LIN {X 0,Y 312.174,Z 269.379,A -85,B 0,C 180,E1 -15950.08,E2 -15950.08} C_VEL
LIN {X 0,Y 314.223,Z 258.273,A -85,B 0,C 180,E1 -15951.484,E2 -15951.484} C_VEL
LIN {X 0,Y 316.003,Z 247.419,A -85,B 0,C 180,E1 -15952.56,E2 -15952.56} C_VEL
LIN {X 0,Y 317.612,Z 235.462,A -85,B 0,C 180,E1 -15953.472,E2 -15953.472} C_VEL
LIN {X 0,Y 318.995,Z 222.423,A -85,B 0,C 180,E1 -15954.183,E2 -15954.183} C_VEL
LIN {X 0,Y 319.798,Z 209.498,A -85,B 0,C 180,E1 -15954.637,E2 -15954.637} C_VEL
LIN {X 0,Y 321.419,Z 151.601,A -85,B 0,C 180,E1 -15955.948,E2 -15955.948} C_VEL
LIN {X 0,Y 317.976,Z 130.29,A -85,B 0,C 180,E1 -15956.843,E2 -15956.843} C_VEL
LIN {X 0,Y 313.089,Z 106.225,A -85,B 0,C 180,E1 -15957.999,E2 -15957.999} C_VEL
LIN {X 0,Y 312.175,Z 103.135,A -85,B 0,C 180,E1 -15958.215,E2 -15958.215} C_VEL
LIN {X 0,Y 309.987,Z 92.53,A -85,B 0,C 180,E1 -15961.43,E2 -15961.43} C_VEL
LIN {X 0,Y 307.446,Z 81.962,A -85,B 0,C 180,E1 -15964.854,E2 -15964.854} C_VEL
LIN {X 0,Y 305.474,Z 74.435,A -85,B 0,C 180,E1 -15967.463,E2 -15967.463} C_VEL
LIN {X 0,Y 305.457,Z 74.429,A -85,B 0,C 180,E1 -15970.6,E2 -15970.6} C_VEL
LIN {X 0,Y 305.428,Z 74.438,A -85,B 0,C 180,E1 -15973.655,E2 -15973.655} C_VEL
LIN {X 0,Y 305.457,Z 74.427,A -85,B 0,C 180,E1 -15977.414,E2 -15977.414} C_VEL
LIN {X 0,Y 305.478,Z 74.431,A -85,B 0,C 180,E1 -15981.598,E2 -15981.598} C_VEL
LIN {X 0,Y 305.465,Z 74.433,A -85,B 0,C 180,E1 -15984.887,E2 -15984.887} C_VEL
LIN {X 0,Y 305.455,Z 74.435,A -85,B 0,C 180,E1 -15988.355,E2 -15988.355} C_VEL
LIN {X 0,Y 305.523,Z 74.424,A -85,B 0,C 180,E1 -15991.114,E2 -15991.114} C_VEL
LIN {X 0,Y 305.574,Z 74.412,A -85,B 0,C 180,E1 -15994.088,E2 -15994.088} C_VEL
LIN {X 0,Y 305.503,Z 74.421,A -85,B 0,C 180,E1 -15998.403,E2 -15998.403} C_VEL
LIN {X 0,Y 305.593,Z 74.417,A -85,B 0,C 180,E1 -16001.218,E2 -16001.218} C_VEL
LIN {X 0,Y 305.652,Z 74.41,A -85,B 0,C 180,E1 -16005.349,E2 -16005.349} C_VEL
LIN {X 0,Y 305.639,Z 74.409,A -85,B 0,C 180,E1 -16009.4,E2 -16009.4} C_VEL
LIN {X 0,Y 305.8,Z 74.385,A -85,B 0,C 180,E1 -16012.074,E2 -16012.074} C_VEL
LIN {X 0,Y 305.687,Z 74.406,A -85,B 0,C 180,E1 -16014.723,E2 -16014.723} C_VEL
LIN {X 0,Y 305.958,Z 74.362,A -85,B 0,C 180,E1 -16018.684,E2 -16018.684} C_VEL
LIN {X 0,Y 305.959,Z 74.374,A -85,B 0,C 180,E1 -16021.316,E2 -16021.316} C_VEL
LIN {X 0,Y 305.684,Z 74.403,A -85,B 0,C 180,E1 -16025.276,E2 -16025.276} C_VEL
LIN {X 0,Y 305.774,Z 74.388,A -85,B 0,C 180,E1 -16027.927,E2 -16027.927} C_VEL
LIN {X 0,Y 305.602,Z 74.416,A -85,B 0,C 180,E1 -16031.945,E2 -16031.945} C_VEL
LIN {X 0,Y 305.611,Z 74.41,A -85,B 0,C 180,E1 -16035.014,E2 -16035.014} C_VEL
LIN {X 0,Y 305.563,Z 74.417,A -85,B 0,C 180,E1 -16039.437,E2 -16039.437} C_VEL
LIN {X 0,Y 305.49,Z 74.424,A -85,B 0,C 180,E1 -16043.04,E2 -16043.04} C_VEL
LIN {X 0,Y 305.48,Z 74.431,A -85,B 0,C 180,E1 -16046.2,E2 -16046.2} C_VEL
LIN {X 0,Y 305.465,Z 74.436,A -85,B 0,C 180,E1 -16049.039,E2 -16049.039} C_VEL
LIN {X 0,Y 305.438,Z 74.437,A -85,B 0,C 180,E1 -16051.953,E2 -16051.953} C_VEL
LIN {X 0,Y 305.463,Z 74.436,A -85,B 0,C 180,E1 -16055.113,E2 -16055.113} C_VEL
LIN {X 0,Y 305.436,Z 74.44,A -85,B 0,C 180,E1 -16058.525,E2 -16058.525} C_VEL
LIN {X 0,Y 305.44,Z 74.426,A -85,B 0,C 180,E1 -16061.857,E2 -16061.857} C_VEL
LIN {X 0,Y 305.401,Z 74.447,A -85,B 0,C 180,E1 -16065.511,E2 -16065.511} C_VEL
LIN {X 0,Y 305.44,Z 74.438,A -85,B 0,C 180,E1 -16068.143,E2 -16068.143} C_VEL
LIN {X 0,Y 305.469,Z 74.592,A -85,B 0,C 180,E1 -16070.734,E2 -16070.734} C_VEL
LIN {X 0,Y 305.694,Z 75.552,A -85,B 0,C 180,E1 -16071.094,E2 -16071.094} C_VEL
LIN {X 0,Y 315.489,Z 94.618,A -85,B 0,C 180,E1 -16072.75,E2 -16072.75} C_VEL
LIN {X 0,Y 322.655,Z 110.769,A -85,B 0,C 180,E1 -16073.933,E2 -16073.933} C_VEL
LIN {X 0,Y 320.349,Z 182.482,A -85,B 0,C 180,E1 -16075.556,E2 -16075.556} C_VEL
LIN {X 0,Y 319.573,Z 195.788,A -85,B 0,C 180,E1 -16076.127,E2 -16076.127} C_VEL
LIN {X 0,Y 318.63,Z 208.433,A -85,B 0,C 180,E1 -16076.947,E2 -16076.947} C_VEL
LIN {X 0,Y 317.275,Z 219.431,A -85,B 0,C 180,E1 -16077.884,E2 -16077.884} C_VEL
LIN {X 0,Y 315.483,Z 231.187,A -85,B 0,C 180,E1 -16079.178,E2 -16079.178} C_VEL
LIN {X 0,Y 313.661,Z 241.965,A -85,B 0,C 180,E1 -16080.695,E2 -16080.695} C_VEL
LIN {X 0,Y 311.646,Z 251.896,A -85,B 0,C 180,E1 -16082.464,E2 -16082.464} C_VEL
LIN {X 0,Y 309.803,Z 260.794,A -85,B 0,C 180,E1 -16084.467,E2 -16084.467} C_VEL
LIN {X 0,Y 308.194,Z 267.818,A -85,B 0,C 180,E1 -16086.48,E2 -16086.48} C_VEL
LIN {X 0,Y 306.828,Z 273.393,A -85,B 0,C 180,E1 -16088.501,E2 -16088.501} C_VEL
LIN {X 0,Y 305.902,Z 277.442,A -85,B 0,C 180,E1 -16090.384,E2 -16090.384} C_VEL
LIN {X 0,Y 304.998,Z 280.942,A -85,B 0,C 180,E1 -16092.569,E2 -16092.569} C_VEL
LIN {X 0,Y 304.582,Z 282.525,A -85,B 0,C 180,E1 -16093.925,E2 -16093.925} C_VEL
LIN {X 0,Y 304.153,Z 284.125,A -85,B 0,C 180,E1 -16096.044,E2 -16096.044} C_VEL
LIN {X 0,Y 303.866,Z 284.702,A -85,B 0,C 180,E1 -16097.986,E2 -16097.986} C_VEL
LIN {X 0,Y 303.732,Z 284.63,A -85,B 0,C 180,E1 -16099.332,E2 -16099.332} C_VEL
LIN {X 0,Y 303.757,Z 284.146,A -85,B 0,C 180,E1 -16100.679,E2 -16100.679} C_VEL
LIN {X 0,Y 303.995,Z 281.922,A -85,B 0,C 180,E1 -16103.362,E2 -16103.362} C_VEL
LIN {X 0,Y 304.17,Z 279.182,A -85,B 0,C 180,E1 -16105.362,E2 -16105.362} C_VEL
LIN {X 0,Y 304.546,Z 275.426,A -85,B 0,C 180,E1 -16107.355,E2 -16107.355} C_VEL
LIN {X 0,Y 304.948,Z 270.574,A -85,B 0,C 180,E1 -16109.34,E2 -16109.34} C_VEL
LIN {X 0,Y 305.686,Z 264.452,A -85,B 0,C 180,E1 -16111.318,E2 -16111.318} C_VEL
LIN {X 0,Y 306.662,Z 256.84,A -85,B 0,C 180,E1 -16113.285,E2 -16113.285} C_VEL
LIN {X 0,Y 307.747,Z 247.299,A -85,B 0,C 180,E1 -16115.241,E2 -16115.241} C_VEL
LIN {X 0,Y 308.92,Z 238.487,A -85,B 0,C 180,E1 -16116.696,E2 -16116.696} C_VEL
LIN {X 0,Y 310.231,Z 227.693,A -85,B 0,C 180,E1 -16118.14,E2 -16118.14} C_VEL
LIN {X 0,Y 311.278,Z 217.16,A -85,B 0,C 180,E1 -16119.257,E2 -16119.257} C_VEL
LIN {X 0,Y 312.202,Z 204.544,A -85,B 0,C 180,E1 -16120.293,E2 -16120.293} C_VEL
LIN {X 0,Y 312.857,Z 191.92,A -85,B 0,C 180,E1 -16121.049,E2 -16121.049} C_VEL
LIN {X 0,Y 313.315,Z 179.752,A -85,B 0,C 180,E1 -16121.524,E2 -16121.524} C_VEL
LIN {X 0,Y 314.897,Z 100.853,A -85,B 0,C 180,E1 -16123.325,E2 -16123.325} C_VEL
LIN {X 0,Y 307.555,Z 79.529,A -85,B 0,C 180,E1 -16124.348,E2 -16124.348} C_VEL
LIN {X 0,Y 305.659,Z 74.413,A -85,B 0,C 180,E1 -16124.624,E2 -16124.624} C_VEL
LIN {X 0,Y 305.591,Z 74.419,A -85,B 0,C 180,E1 -16128.783,E2 -16128.783} C_VEL
LIN {X 0,Y 305.487,Z 74.43,A -85,B 0,C 180,E1 -16133.04,E2 -16133.04} C_VEL
LIN {X 0,Y 305.548,Z 74.427,A -85,B 0,C 180,E1 -16136.227,E2 -16136.227} C_VEL
LIN {X 0,Y 305.489,Z 74.43,A -85,B 0,C 180,E1 -16139.048,E2 -16139.048} C_VEL
LIN {X 0,Y 305.445,Z 74.44,A -85,B 0,C 180,E1 -16141.952,E2 -16141.952} C_VEL
LIN {X 0,Y 305.465,Z 74.433,A -85,B 0,C 180,E1 -16145.113,E2 -16145.113} C_VEL
LIN {X 0,Y 305.469,Z 74.432,A -85,B 0,C 180,E1 -16148.533,E2 -16148.533} C_VEL
LIN {X 0,Y 305.475,Z 74.431,A -85,B 0,C 180,E1 -16152.59,E2 -16152.59} C_VEL
LIN {X 0,Y 305.457,Z 74.438,A -85,B 0,C 180,E1 -16157.415,E2 -16157.415} C_VEL
LIN {X 0,Y 305.442,Z 74.436,A -85,B 0,C 180,E1 -16159.149,E2 -16159.149} C_VEL
LIN {X 0,Y 304.808,Z 74.519,A -85,B 0,C 180,E1 -16160.25,E2 -16160.25} C_VEL
LIN {X 0,Y 301.942,Z 74.872,A -85,B 0,C 180,E1 -16162.043,E2 -16162.043} C_VEL
LIN {X 0,Y 299.502,Z 75.176,A -85,B 0,C 180,E1 -16163.497,E2 -16163.497} C_VEL
LIN {X 0,Y 298.474,Z 75.302,A -85,B 0,C 180,E1 -16164.624,E2 -16164.624} C_VEL
LIN {X 0,Y 298.402,Z 75.309,A -85,B 0,C 180,E1 -16165.006,E2 -16165.006} C_VEL
LIN {X 0,Y 298.395,Z 75.316,A -85,B 0,C 180,E1 -16168.791,E2 -16168.791} C_VEL
LIN {X 0,Y 298.462,Z 75.305,A -85,B 0,C 180,E1 -16171.904,E2 -16171.904} C_VEL
LIN {X 0,Y 298.489,Z 75.304,A -85,B 0,C 180,E1 -16174.924,E2 -16174.924} C_VEL
LIN {X 0,Y 298.454,Z 75.305,A -85,B 0,C 180,E1 -16179.316,E2 -16179.316} C_VEL
LIN {X 0,Y 298.541,Z 75.293,A -85,B 0,C 180,E1 -16182.18,E2 -16182.18} C_VEL
LIN {X 0,Y 298.597,Z 75.284,A -85,B 0,C 180,E1 -16184.995,E2 -16184.995} C_VEL
LIN {X 0,Y 298.587,Z 75.289,A -85,B 0,C 180,E1 -16189.147,E2 -16189.147} C_VEL
LIN {X 0,Y 298.736,Z 75.273,A -85,B 0,C 180,E1 -16191.885,E2 -16191.885} C_VEL
LIN {X 0,Y 298.657,Z 75.273,A -85,B 0,C 180,E1 -16194.599,E2 -16194.599} C_VEL
LIN {X 0,Y 298.926,Z 75.245,A -85,B 0,C 180,E1 -16198.653,E2 -16198.653} C_VEL
LIN {X 0,Y 298.926,Z 75.248,A -85,B 0,C 180,E1 -16201.347,E2 -16201.347} C_VEL
LIN {X 0,Y 298.643,Z 75.283,A -85,B 0,C 180,E1 -16205.402,E2 -16205.402} C_VEL
LIN {X 0,Y 298.712,Z 75.274,A -85,B 0,C 180,E1 -16208.116,E2 -16208.116} C_VEL
LIN {X 0,Y 298.554,Z 75.293,A -85,B 0,C 180,E1 -16212.232,E2 -16212.232} C_VEL
LIN {X 0,Y 298.553,Z 75.297,A -85,B 0,C 180,E1 -16215.169,E2 -16215.169} C_VEL
LIN {X 0,Y 298.524,Z 75.3,A -85,B 0,C 180,E1 -16219.244,E2 -16219.244} C_VEL
LIN {X 0,Y 298.429,Z 75.31,A -85,B 0,C 180,E1 -16223.6,E2 -16223.6} C_VEL
LIN {X 0,Y 298.42,Z 75.313,A -85,B 0,C 180,E1 -16226.581,E2 -16226.581} C_VEL
LIN {X 0,Y 298.403,Z 75.313,A -85,B 0,C 180,E1 -16229.643,E2 -16229.643} C_VEL
LIN {X 0,Y 298.396,Z 75.318,A -85,B 0,C 180,E1 -16232.8,E2 -16232.8} C_VEL
LIN {X 0,Y 298.45,Z 75.31,A -85,B 0,C 180,E1 -16236.808,E2 -16236.808} C_VEL
LIN {X 0,Y 298.39,Z 75.315,A -85,B 0,C 180,E1 -16241.088,E2 -16241.088} C_VEL
LIN {X 0,Y 298.401,Z 75.312,A -85,B 0,C 180,E1 -16243.103,E2 -16243.103} C_VEL
LIN {X 0,Y 298.406,Z 75.313,A -85,B 0,C 180,E1 -16246.921,E2 -16246.921} C_VEL
LIN {X 0,Y 298.398,Z 75.314,A -85,B 0,C 180,E1 -16251.008,E2 -16251.008} C_VEL
LIN {X 0,Y 298.419,Z 75.312,A -85,B 0,C 180,E1 -16253.93,E2 -16253.93} C_VEL
LIN {X 0,Y 298.459,Z 75.446,A -85,B 0,C 180,E1 -16257.157,E2 -16257.157} C_VEL
LIN {X 0,Y 301.343,Z 88.771,A -85,B 0,C 180,E1 -16261.057,E2 -16261.057} C_VEL
LIN {X 0,Y 302.506,Z 95.962,A -85,B 0,C 180,E1 -16263.061,E2 -16263.061} C_VEL
LIN {X 0,Y 301.566,Z 103.824,A -85,B 0,C 180,E1 -16265.076,E2 -16265.076} C_VEL
LIN {X 0,Y 306.342,Z 141.137,A -85,B 0,C 180,E1 -16266.335,E2 -16266.335} C_VEL
LIN {X 0,Y 307.368,Z 151.276,A -85,B 0,C 180,E1 -16266.651,E2 -16266.651} C_VEL
LIN {X 0,Y 306.075,Z 212.628,A -85,B 0,C 180,E1 -16268.091,E2 -16268.091} C_VEL
LIN {X 0,Y 305.295,Z 225.998,A -85,B 0,C 180,E1 -16268.653,E2 -16268.653} C_VEL
LIN {X 0,Y 304.267,Z 238.814,A -85,B 0,C 180,E1 -16269.463,E2 -16269.463} C_VEL
LIN {X 0,Y 302.972,Z 250.972,A -85,B 0,C 180,E1 -16270.521,E2 -16270.521} C_VEL
LIN {X 0,Y 301.528,Z 262.552,A -85,B 0,C 180,E1 -16271.835,E2 -16271.835} C_VEL
LIN {X 0,Y 300.343,Z 273.016,A -85,B 0,C 180,E1 -16273.342,E2 -16273.342} C_VEL
LIN {X 0,Y 299.404,Z 281.24,A -85,B 0,C 180,E1 -16274.799,E2 -16274.799} C_VEL
LIN {X 0,Y 298.344,Z 290.113,A -85,B 0,C 180,E1 -16276.722,E2 -16276.722} C_VEL
LIN {X 0,Y 297.419,Z 297.659,A -85,B 0,C 180,E1 -16278.758,E2 -16278.758} C_VEL
LIN {X 0,Y 296.928,Z 304.631,A -85,B 0,C 180,E1 -16281.15,E2 -16281.15} C_VEL
LIN {X 0,Y 296.642,Z 309.207,A -85,B 0,C 180,E1 -16283.197,E2 -16283.197} C_VEL
LIN {X 0,Y 296.641,Z 311.618,A -85,B 0,C 180,E1 -16284.562,E2 -16284.562} C_VEL
LIN {X 0,Y 296.692,Z 313.588,A -85,B 0,C 180,E1 -16285.925,E2 -16285.925} C_VEL
LIN {X 0,Y 296.691,Z 315.127,A -85,B 0,C 180,E1 -16287.284,E2 -16287.284} C_VEL
LIN {X 0,Y 296.759,Z 316.208,A -85,B 0,C 180,E1 -16288.643,E2 -16288.643} C_VEL
LIN {X 0,Y 296.843,Z 316.882,A -85,B 0,C 180,E1 -16290,E2 -16290} C_VEL
LIN {X 0,Y 296.624,Z 317.031,A -85,B 0,C 180,E1 -16292.716,E2 -16292.716} C_VEL
LIN {X 0,Y 296.597,Z 316.486,A -85,B 0,C 180,E1 -16294.076,E2 -16294.076} C_VEL
LIN {X 0,Y 296.646,Z 314.191,A -85,B 0,C 180,E1 -16296.803,E2 -16296.803} C_VEL
LIN {X 0,Y 296.972,Z 311.382,A -85,B 0,C 180,E1 -16298.849,E2 -16298.849} C_VEL
LIN {X 0,Y 297.529,Z 307.567,A -85,B 0,C 180,E1 -16300.893,E2 -16300.893} C_VEL
LIN {X 0,Y 298.461,Z 302.656,A -85,B 0,C 180,E1 -16302.926,E2 -16302.926} C_VEL
LIN {X 0,Y 299.869,Z 296.503,A -85,B 0,C 180,E1 -16304.94,E2 -16304.94} C_VEL
LIN {X 0,Y 301.468,Z 289.016,A -85,B 0,C 180,E1 -16306.909,E2 -16306.909} C_VEL
LIN {X 0,Y 303.08,Z 281.127,A -85,B 0,C 180,E1 -16308.593,E2 -16308.593} C_VEL
LIN {X 0,Y 305.307,Z 270.619,A -85,B 0,C 180,E1 -16310.375,E2 -16310.375} C_VEL
LIN {X 0,Y 307.451,Z 259.953,A -85,B 0,C 180,E1 -16311.806,E2 -16311.806} C_VEL
LIN {X 0,Y 309.207,Z 249.659,A -85,B 0,C 180,E1 -16312.907,E2 -16312.907} C_VEL
LIN {X 0,Y 311.029,Z 237.375,A -85,B 0,C 180,E1 -16313.911,E2 -16313.911} C_VEL
LIN {X 0,Y 312.502,Z 224.487,A -85,B 0,C 180,E1 -16314.674,E2 -16314.674} C_VEL
LIN {X 0,Y 313.425,Z 212.064,A -85,B 0,C 180,E1 -16315.172,E2 -16315.172} C_VEL
LIN {X 0,Y 315.209,Z 152.445,A -85,B 0,C 180,E1 -16316.561,E2 -16316.561} C_VEL
LIN {X 0,Y 311.622,Z 130.195,A -85,B 0,C 180,E1 -16317.528,E2 -16317.528} C_VEL
LIN {X 0,Y 307.049,Z 108.021,A -85,B 0,C 180,E1 -16318.641,E2 -16318.641} C_VEL
LIN {X 0,Y 304.973,Z 102.645,A -85,B 0,C 180,E1 -16319.07,E2 -16319.07} C_VEL
LIN {X 0,Y 302.402,Z 90.76,A -85,B 0,C 180,E1 -16322.837,E2 -16322.837} C_VEL
LIN {X 0,Y 299.638,Z 79.777,A -85,B 0,C 180,E1 -16326.594,E2 -16326.594} C_VEL
LIN {X 0,Y 298.449,Z 75.301,A -85,B 0,C 180,E1 -16328.288,E2 -16328.288} C_VEL
LIN {X 0,Y 298.387,Z 75.316,A -85,B 0,C 180,E1 -16331.261,E2 -16331.261} C_VEL
LIN {X 0,Y 298.356,Z 75.312,A -85,B 0,C 180,E1 -16335.035,E2 -16335.035} C_VEL
LIN {X 0,Y 298.387,Z 75.312,A -85,B 0,C 180,E1 -16338.738,E2 -16338.738} C_VEL
LIN {X 0,Y 298.416,Z 75.307,A -85,B 0,C 180,E1 -16342.242,E2 -16342.242} C_VEL
LIN {X 0,Y 298.411,Z 75.308,A -85,B 0,C 180,E1 -16345.581,E2 -16345.581} C_VEL
LIN {X 0,Y 298.398,Z 75.316,A -85,B 0,C 180,E1 -16348.791,E2 -16348.791} C_VEL
LIN {X 0,Y 298.466,Z 75.306,A -85,B 0,C 180,E1 -16351.904,E2 -16351.904} C_VEL
LIN {X 0,Y 298.489,Z 75.298,A -85,B 0,C 180,E1 -16354.924,E2 -16354.924} C_VEL
LIN {X 0,Y 298.453,Z 75.304,A -85,B 0,C 180,E1 -16359.315,E2 -16359.315} C_VEL
LIN {X 0,Y 298.541,Z 75.29,A -85,B 0,C 180,E1 -16362.179,E2 -16362.179} C_VEL
LIN {X 0,Y 298.597,Z 75.29,A -85,B 0,C 180,E1 -16364.995,E2 -16364.995} C_VEL
LIN {X 0,Y 298.595,Z 75.287,A -85,B 0,C 180,E1 -16369.147,E2 -16369.147} C_VEL
LIN {X 0,Y 298.744,Z 75.266,A -85,B 0,C 180,E1 -16371.885,E2 -16371.885} C_VEL
LIN {X 0,Y 298.658,Z 75.28,A -85,B 0,C 180,E1 -16374.599,E2 -16374.599} C_VEL
LIN {X 0,Y 298.925,Z 75.237,A -85,B 0,C 180,E1 -16378.653,E2 -16378.653} C_VEL
LIN {X 0,Y 298.925,Z 75.25,A -85,B 0,C 180,E1 -16381.347,E2 -16381.347} C_VEL
LIN {X 0,Y 298.778,Z 75.267,A -85,B 0,C 180,E1 -16386.754,E2 -16386.754} C_VEL
LIN {X 0,Y 298.628,Z 75.276,A -85,B 0,C 180,E1 -16389.482,E2 -16389.482} C_VEL
LIN {X 0,Y 298.548,Z 75.285,A -85,B 0,C 180,E1 -16393.615,E2 -16393.615} C_VEL
LIN {X 0,Y 298.49,Z 75.303,A -85,B 0,C 180,E1 -16396.412,E2 -16396.412} C_VEL
LIN {X 0,Y 298.501,Z 75.298,A -85,B 0,C 180,E1 -16399.648,E2 -16399.648} C_VEL
LIN {X 0,Y 298.428,Z 75.305,A -85,B 0,C 180,E1 -16403.6,E2 -16403.6} C_VEL
LIN {X 0,Y 298.418,Z 75.307,A -85,B 0,C 180,E1 -16406.581,E2 -16406.581} C_VEL
LIN {X 0,Y 298.401,Z 75.314,A -85,B 0,C 180,E1 -16409.643,E2 -16409.643} C_VEL
LIN {X 0,Y 298.394,Z 75.315,A -85,B 0,C 180,E1 -16412.8,E2 -16412.8} C_VEL
LIN {X 0,Y 298.429,Z 75.307,A -85,B 0,C 180,E1 -16416.803,E2 -16416.803} C_VEL
LIN {X 0,Y 298.386,Z 75.299,A -85,B 0,C 180,E1 -16421.087,E2 -16421.087} C_VEL
LIN {X 0,Y 298.399,Z 75.318,A -85,B 0,C 180,E1 -16423.103,E2 -16423.103} C_VEL
LIN {X 0,Y 298.403,Z 75.317,A -85,B 0,C 180,E1 -16426.921,E2 -16426.921} C_VEL
LIN {X 0,Y 298.442,Z 75.344,A -85,B 0,C 180,E1 -16429.955,E2 -16429.955} C_VEL
LIN {X 0,Y 298.551,Z 76.08,A -85,B 0,C 180,E1 -16430.207,E2 -16430.207} C_VEL
LIN {X 0,Y 299.83,Z 78.759,A -85,B 0,C 180,E1 -16430.448,E2 -16430.448} C_VEL
LIN {X 0,Y 306.364,Z 90.758,A -85,B 0,C 180,E1 -16431.592,E2 -16431.592} C_VEL
LIN {X 0,Y 314.302,Z 107.493,A -85,B 0,C 180,E1 -16432.956,E2 -16432.956} C_VEL
LIN {X 0,Y 316.501,Z 112.872,A -85,B 0,C 180,E1 -16433.337,E2 -16433.337} C_VEL
LIN {X 0,Y 314.165,Z 182.264,A -85,B 0,C 180,E1 -16434.925,E2 -16434.925} C_VEL
LIN {X 0,Y 313.406,Z 194.984,A -85,B 0,C 180,E1 -16435.464,E2 -16435.464} C_VEL
LIN {X 0,Y 312.466,Z 207.132,A -85,B 0,C 180,E1 -16436.236,E2 -16436.236} C_VEL
LIN {X 0,Y 311.086,Z 218.328,A -85,B 0,C 180,E1 -16437.166,E2 -16437.166} C_VEL
LIN {X 0,Y 309.481,Z 229.094,A -85,B 0,C 180,E1 -16438.322,E2 -16438.322} C_VEL
LIN {X 0,Y 307.565,Z 240.054,A -85,B 0,C 180,E1 -16439.82,E2 -16439.82} C_VEL
LIN {X 0,Y 305.568,Z 249.853,A -85,B 0,C 180,E1 -16441.494,E2 -16441.494} C_VEL
LIN {X 0,Y 303.844,Z 257.821,A -85,B 0,C 180,E1 -16443.189,E2 -16443.189} C_VEL
LIN {X 0,Y 302.038,Z 265.527,A -85,B 0,C 180,E1 -16445.239,E2 -16445.239} C_VEL
LIN {X 0,Y 300.484,Z 271.67,A -85,B 0,C 180,E1 -16447.299,E2 -16447.299} C_VEL
LIN {X 0,Y 299.289,Z 276.492,A -85,B 0,C 180,E1 -16449.376,E2 -16449.376} C_VEL
LIN {X 0,Y 298.369,Z 280.149,A -85,B 0,C 180,E1 -16451.459,E2 -16451.459} C_VEL
LIN {X 0,Y 297.612,Z 282.751,A -85,B 0,C 180,E1 -16453.538,E2 -16453.538} C_VEL
LIN {X 0,Y 297.104,Z 284.53,A -85,B 0,C 180,E1 -16455.896,E2 -16455.896} C_VEL
LIN {X 0,Y 296.835,Z 285.072,A -85,B 0,C 180,E1 -16457.697,E2 -16457.697} C_VEL
LIN {X 0,Y 296.652,Z 284.609,A -85,B 0,C 180,E1 -16460.454,E2 -16460.454} C_VEL
LIN {X 0,Y 296.728,Z 283.745,A -85,B 0,C 180,E1 -16461.83,E2 -16461.83} C_VEL
LIN {X 0,Y 296.993,Z 281.98,A -85,B 0,C 180,E1 -16463.658,E2 -16463.658} C_VEL
LIN {X 0,Y 297.122,Z 278.725,A -85,B 0,C 180,E1 -16465.931,E2 -16465.931} C_VEL
LIN {X 0,Y 297.589,Z 274.69,A -85,B 0,C 180,E1 -16467.97,E2 -16467.97} C_VEL
LIN {X 0,Y 298.192,Z 268.515,A -85,B 0,C 180,E1 -16470.338,E2 -16470.338} C_VEL
LIN {X 0,Y 299.15,Z 261.775,A -85,B 0,C 180,E1 -16472.356,E2 -16472.356} C_VEL
LIN {X 0,Y 300.146,Z 253.433,A -85,B 0,C 180,E1 -16474.365,E2 -16474.365} C_VEL
LIN {X 0,Y 301.166,Z 244.842,A -85,B 0,C 180,E1 -16476.028,E2 -16476.028} C_VEL
LIN {X 0,Y 302.694,Z 234.206,A -85,B 0,C 180,E1 -16477.672,E2 -16477.672} C_VEL
LIN {X 0,Y 303.852,Z 223.677,A -85,B 0,C 180,E1 -16478.982,E2 -16478.982} C_VEL
LIN {X 0,Y 304.911,Z 211.957,A -85,B 0,C 180,E1 -16480.123,E2 -16480.123} C_VEL
LIN {X 0,Y 305.804,Z 198.526,A -85,B 0,C 180,E1 -16481.097,E2 -16481.097} C_VEL
LIN {X 0,Y 306.404,Z 185.409,A -85,B 0,C 180,E1 -16481.746,E2 -16481.746} C_VEL
LIN {X 0,Y 306.876,Z 168.023,A -85,B 0,C 180,E1 -16482.226,E2 -16482.226} C_VEL
LIN {X 0,Y 308.182,Z 102.089,A -85,B 0,C 180,E1 -16483.75,E2 -16483.75} C_VEL
LIN {X 0,Y 300.981,Z 81.491,A -85,B 0,C 180,E1 -16484.779,E2 -16484.779} C_VEL
LIN {X 0,Y 298.658,Z 75.723,A -85,B 0,C 180,E1 -16485.1,E2 -16485.1} C_VEL
LIN {X 0,Y 298.582,Z 75.293,A -85,B 0,C 180,E1 -16485.192,E2 -16485.192} C_VEL
LIN {X 0,Y 298.54,Z 75.296,A -85,B 0,C 180,E1 -16489.243,E2 -16489.243} C_VEL
LIN {X 0,Y 298.43,Z 75.309,A -85,B 0,C 180,E1 -16493.6,E2 -16493.6} C_VEL
LIN {X 0,Y 298.49,Z 75.303,A -85,B 0,C 180,E1 -16496.575,E2 -16496.575} C_VEL
LIN {X 0,Y 298.418,Z 75.313,A -85,B 0,C 180,E1 -16499.642,E2 -16499.642} C_VEL
LIN {X 0,Y 298.397,Z 75.313,A -85,B 0,C 180,E1 -16502.8,E2 -16502.8} C_VEL
LIN {X 0,Y 298.466,Z 75.304,A -85,B 0,C 180,E1 -16506.813,E2 -16506.813} C_VEL
LIN {X 0,Y 298.414,Z 75.311,A -85,B 0,C 180,E1 -16511.094,E2 -16511.094} C_VEL
LIN {X 0,Y 298.356,Z 75.319,A -85,B 0,C 180,E1 -16515.035,E2 -16515.035} C_VEL
LIN {X 0,Y 298.386,Z 75.314,A -85,B 0,C 180,E1 -16518.739,E2 -16518.739} C_VEL
LIN {X 0,Y 298.416,Z 75.31,A -85,B 0,C 180,E1 -16522.242,E2 -16522.242} C_VEL
LIN {X 0,Y 298.402,Z 75.309,A -85,B 0,C 180,E1 -16525.006,E2 -16525.006} C_VEL
LIN {X 0,Y 297.763,Z 75.393,A -85,B 0,C 180,E1 -16526.131,E2 -16526.131} C_VEL
LIN {X 0,Y 294.909,Z 75.747,A -85,B 0,C 180,E1 -16527.963,E2 -16527.963} C_VEL
LIN {X 0,Y 292.48,Z 76.049,A -85,B 0,C 180,E1 -16529.45,E2 -16529.45} C_VEL
LIN {X 0,Y 291.452,Z 76.178,A -85,B 0,C 180,E1 -16530.603,E2 -16530.603} C_VEL
LIN {X 0,Y 291.377,Z 76.189,A -85,B 0,C 180,E1 -16530.993,E2 -16530.993} C_VEL
LIN {X 0,Y 291.417,Z 76.183,A -85,B 0,C 180,E1 -16534.272,E2 -16534.272} C_VEL
LIN {X 0,Y 291.385,Z 76.187,A -85,B 0,C 180,E1 -16537.3,E2 -16537.3} C_VEL
LIN {X 0,Y 291.462,Z 76.179,A -85,B 0,C 180,E1 -16540.271,E2 -16540.271} C_VEL
LIN {X 0,Y 291.559,Z 76.16,A -85,B 0,C 180,E1 -16544.624,E2 -16544.624} C_VEL
LIN {X 0,Y 291.533,Z 76.169,A -85,B 0,C 180,E1 -16548.881,E2 -16548.881} C_VEL
LIN {X 0,Y 291.684,Z 76.15,A -85,B 0,C 180,E1 -16551.688,E2 -16551.688} C_VEL
LIN {X 0,Y 291.628,Z 76.148,A -85,B 0,C 180,E1 -16554.468,E2 -16554.468} C_VEL
LIN {X 0,Y 291.892,Z 76.121,A -85,B 0,C 180,E1 -16558.621,E2 -16558.621} C_VEL
LIN {X 0,Y 291.893,Z 76.125,A -85,B 0,C 180,E1 -16561.38,E2 -16561.38} C_VEL
LIN {X 0,Y 291.612,Z 76.16,A -85,B 0,C 180,E1 -16565.532,E2 -16565.532} C_VEL
LIN {X 0,Y 291.676,Z 76.151,A -85,B 0,C 180,E1 -16568.917,E2 -16568.917} C_VEL
LIN {X 0,Y 291.521,Z 76.17,A -85,B 0,C 180,E1 -16572.531,E2 -16572.531} C_VEL
LIN {X 0,Y 291.51,Z 76.173,A -85,B 0,C 180,E1 -16575.379,E2 -16575.379} C_VEL
LIN {X 0,Y 291.454,Z 76.177,A -85,B 0,C 180,E1 -16579.875,E2 -16579.875} C_VEL
LIN {X 0,Y 291.371,Z 76.189,A -85,B 0,C 180,E1 -16584.208,E2 -16584.208} C_VEL
LIN {X 0,Y 291.365,Z 76.192,A -85,B 0,C 180,E1 -16587.278,E2 -16587.278} C_VEL
LIN {X 0,Y 291.325,Z 76.197,A -85,B 0,C 180,E1 -16590.438,E2 -16590.438} C_VEL
LIN {X 0,Y 291.347,Z 76.192,A -85,B 0,C 180,E1 -16593.698,E2 -16593.698} C_VEL
LIN {X 0,Y 291.379,Z 76.188,A -85,B 0,C 180,E1 -16597.254,E2 -16597.254} C_VEL
LIN {X 0,Y 291.336,Z 76.196,A -85,B 0,C 180,E1 -16600.642,E2 -16600.642} C_VEL
LIN {X 0,Y 291.293,Z 76.202,A -85,B 0,C 180,E1 -16604.402,E2 -16604.402} C_VEL
LIN {X 0,Y 291.328,Z 76.198,A -85,B 0,C 180,E1 -16608.404,E2 -16608.404} C_VEL
LIN {X 0,Y 291.347,Z 76.193,A -85,B 0,C 180,E1 -16611.157,E2 -16611.157} C_VEL
LIN {X 0,Y 291.363,Z 76.192,A -85,B 0,C 180,E1 -16614.626,E2 -16614.626} C_VEL
LIN {X 0,Y 291.41,Z 76.315,A -85,B 0,C 180,E1 -16616.752,E2 -16616.752} C_VEL
LIN {X 0,Y 294.22,Z 89.361,A -85,B 0,C 180,E1 -16620.68,E2 -16620.68} C_VEL
LIN {X 0,Y 295.527,Z 96.631,A -85,B 0,C 180,E1 -16622.77,E2 -16622.77} C_VEL
LIN {X 0,Y 294.778,Z 103.429,A -85,B 0,C 180,E1 -16624.562,E2 -16624.562} C_VEL
LIN {X 0,Y 299.245,Z 138.132,A -85,B 0,C 180,E1 -16625.777,E2 -16625.777} C_VEL
LIN {X 0,Y 300.648,Z 152.164,A -85,B 0,C 180,E1 -16626.225,E2 -16626.225} C_VEL
LIN {X 0,Y 299.32,Z 212.635,A -85,B 0,C 180,E1 -16627.681,E2 -16627.681} C_VEL
LIN {X 0,Y 298.499,Z 226.305,A -85,B 0,C 180,E1 -16628.279,E2 -16628.279} C_VEL
LIN {X 0,Y 297.48,Z 238.371,A -85,B 0,C 180,E1 -16629.063,E2 -16629.063} C_VEL
LIN {X 0,Y 296.276,Z 249.754,A -85,B 0,C 180,E1 -16630.062,E2 -16630.062} C_VEL
LIN {X 0,Y 294.785,Z 261.491,A -85,B 0,C 180,E1 -16631.405,E2 -16631.405} C_VEL
LIN {X 0,Y 293.494,Z 272.069,A -85,B 0,C 180,E1 -16632.942,E2 -16632.942} C_VEL
LIN {X 0,Y 292.473,Z 280.169,A -85,B 0,C 180,E1 -16634.388,E2 -16634.388} C_VEL
LIN {X 0,Y 291.489,Z 287.915,A -85,B 0,C 180,E1 -16636.048,E2 -16636.048} C_VEL
LIN {X 0,Y 290.702,Z 294.633,A -85,B 0,C 180,E1 -16637.787,E2 -16637.787} C_VEL
LIN {X 0,Y 290.141,Z 300.221,A -85,B 0,C 180,E1 -16639.533,E2 -16639.533} C_VEL
LIN {X 0,Y 289.753,Z 305.679,A -85,B 0,C 180,E1 -16641.632,E2 -16641.632} C_VEL
LIN {X 0,Y 289.541,Z 310.05,A -85,B 0,C 180,E1 -16643.799,E2 -16643.799} C_VEL
LIN {X 0,Y 289.601,Z 313.09,A -85,B 0,C 180,E1 -16645.825,E2 -16645.825} C_VEL
LIN {X 0,Y 289.612,Z 314.654,A -85,B 0,C 180,E1 -16647.218,E2 -16647.218} C_VEL
LIN {X 0,Y 289.665,Z 315.773,A -85,B 0,C 180,E1 -16648.61,E2 -16648.61} C_VEL
LIN {X 0,Y 289.752,Z 316.467,A -85,B 0,C 180,E1 -16650,E2 -16650} C_VEL
LIN {X 0,Y 289.545,Z 316.657,A -85,B 0,C 180,E1 -16652.782,E2 -16652.782} C_VEL
LIN {X 0,Y 289.51,Z 316.15,A -85,B 0,C 180,E1 -16654.176,E2 -16654.176} C_VEL
LIN {X 0,Y 289.571,Z 313.898,A -85,B 0,C 180,E1 -16656.97,E2 -16656.97} C_VEL
LIN {X 0,Y 289.911,Z 311.133,A -85,B 0,C 180,E1 -16659.066,E2 -16659.066} C_VEL
LIN {X 0,Y 290.501,Z 307.365,A -85,B 0,C 180,E1 -16661.16,E2 -16661.16} C_VEL
LIN {X 0,Y 291.532,Z 302.505,A -85,B 0,C 180,E1 -16663.239,E2 -16663.239} C_VEL
LIN {X 0,Y 292.974,Z 296.407,A -85,B 0,C 180,E1 -16665.3,E2 -16665.3} C_VEL
LIN {X 0,Y 294.8,Z 288.136,A -85,B 0,C 180,E1 -16667.522,E2 -16667.522} C_VEL
LIN {X 0,Y 296.726,Z 279.436,A -85,B 0,C 180,E1 -16669.365,E2 -16669.365} C_VEL
LIN {X 0,Y 299.135,Z 268.654,A -85,B 0,C 180,E1 -16671.176,E2 -16671.176} C_VEL
LIN {X 0,Y 301.31,Z 257.57,A -85,B 0,C 180,E1 -16672.635,E2 -16672.635} C_VEL
LIN {X 0,Y 303.542,Z 244.97,A -85,B 0,C 180,E1 -16673.903,E2 -16673.903} C_VEL
LIN {X 0,Y 305.32,Z 232.457,A -85,B 0,C 180,E1 -16674.84,E2 -16674.84} C_VEL
LIN {X 0,Y 306.672,Z 219.115,A -85,B 0,C 180,E1 -16675.539,E2 -16675.539} C_VEL
LIN {X 0,Y 307.571,Z 205.376,A -85,B 0,C 180,E1 -16675.977,E2 -16675.977} C_VEL
LIN {X 0,Y 308.985,Z 152.995,A -85,B 0,C 180,E1 -16677.213,E2 -16677.213} C_VEL
LIN {X 0,Y 305.669,Z 132.107,A -85,B 0,C 180,E1 -16678.148,E2 -16678.148} C_VEL
LIN {X 0,Y 301.282,Z 110.567,A -85,B 0,C 180,E1 -16679.262,E2 -16679.262} C_VEL
LIN {X 0,Y 297.649,Z 102.186,A -85,B 0,C 180,E1 -16679.987,E2 -16679.987} C_VEL
LIN {X 0,Y 295.584,Z 92.497,A -85,B 0,C 180,E1 -16683.152,E2 -16683.152} C_VEL
LIN {X 0,Y 292.949,Z 81.973,A -85,B 0,C 180,E1 -16686.853,E2 -16686.853} C_VEL
LIN {X 0,Y 291.362,Z 76.177,A -85,B 0,C 180,E1 -16689.081,E2 -16689.081} C_VEL
LIN {X 0,Y 291.322,Z 76.191,A -85,B 0,C 180,E1 -16692.492,E2 -16692.492} C_VEL
LIN {X 0,Y 291.311,Z 76.193,A -85,B 0,C 180,E1 -16696.366,E2 -16696.366} C_VEL
LIN {X 0,Y 291.384,Z 76.179,A -85,B 0,C 180,E1 -16700.518,E2 -16700.518} C_VEL
LIN {X 0,Y 291.41,Z 76.177,A -85,B 0,C 180,E1 -16702.92,E2 -16702.92} C_VEL
LIN {X 0,Y 291.347,Z 76.185,A -85,B 0,C 180,E1 -16706.302,E2 -16706.302} C_VEL
LIN {X 0,Y 291.39,Z 76.18,A -85,B 0,C 180,E1 -16710.26,E2 -16710.26} C_VEL
LIN {X 0,Y 291.419,Z 76.175,A -85,B 0,C 180,E1 -16714.272,E2 -16714.272} C_VEL
LIN {X 0,Y 291.385,Z 76.183,A -85,B 0,C 180,E1 -16717.3,E2 -16717.3} C_VEL
LIN {X 0,Y 291.46,Z 76.178,A -85,B 0,C 180,E1 -16720.27,E2 -16720.27} C_VEL
LIN {X 0,Y 291.558,Z 76.165,A -85,B 0,C 180,E1 -16724.624,E2 -16724.624} C_VEL
LIN {X 0,Y 291.539,Z 76.163,A -85,B 0,C 180,E1 -16728.881,E2 -16728.881} C_VEL
LIN {X 0,Y 291.691,Z 76.147,A -85,B 0,C 180,E1 -16731.688,E2 -16731.688} C_VEL
LIN {X 0,Y 291.628,Z 76.154,A -85,B 0,C 180,E1 -16734.468,E2 -16734.468} C_VEL
LIN {X 0,Y 291.891,Z 76.113,A -85,B 0,C 180,E1 -16738.62,E2 -16738.62} C_VEL
LIN {X 0,Y 291.891,Z 76.127,A -85,B 0,C 180,E1 -16741.38,E2 -16741.38} C_VEL
LIN {X 0,Y 291.725,Z 76.146,A -85,B 0,C 180,E1 -16746.918,E2 -16746.918} C_VEL
LIN {X 0,Y 291.57,Z 76.157,A -85,B 0,C 180,E1 -16749.714,E2 -16749.714} C_VEL
LIN {X 0,Y 291.518,Z 76.16,A -85,B 0,C 180,E1 -16753.95,E2 -16753.95} C_VEL
LIN {X 0,Y 291.45,Z 76.172,A -85,B 0,C 180,E1 -16758.269,E2 -16758.269} C_VEL
LIN {X 0,Y 291.376,Z 76.19,A -85,B 0,C 180,E1 -16761.211,E2 -16761.211} C_VEL
LIN {X 0,Y 291.37,Z 76.187,A -85,B 0,C 180,E1 -16764.208,E2 -16764.208} C_VEL
LIN {X 0,Y 291.364,Z 76.184,A -85,B 0,C 180,E1 -16767.277,E2 -16767.277} C_VEL
LIN {X 0,Y 291.323,Z 76.191,A -85,B 0,C 180,E1 -16770.438,E2 -16770.438} C_VEL
LIN {X 0,Y 291.345,Z 76.189,A -85,B 0,C 180,E1 -16773.698,E2 -16773.698} C_VEL
LIN {X 0,Y 291.361,Z 76.188,A -85,B 0,C 180,E1 -16777.249,E2 -16777.249} C_VEL
LIN {X 0,Y 291.331,Z 76.178,A -85,B 0,C 180,E1 -16780.643,E2 -16780.643} C_VEL
LIN {X 0,Y 291.291,Z 76.201,A -85,B 0,C 180,E1 -16784.402,E2 -16784.402} C_VEL
LIN {X 0,Y 291.327,Z 76.197,A -85,B 0,C 180,E1 -16788.404,E2 -16788.404} C_VEL
LIN {X 0,Y 291.387,Z 76.38,A -85,B 0,C 180,E1 -16789.24,E2 -16789.24} C_VEL
LIN {X 0,Y 292.51,Z 79.277,A -85,B 0,C 180,E1 -16789.495,E2 -16789.495} C_VEL
LIN {X 0,Y 294.006,Z 81.582,A -85,B 0,C 180,E1 -16789.765,E2 -16789.765} C_VEL
LIN {X 0,Y 300.332,Z 93.086,A -85,B 0,C 180,E1 -16790.917,E2 -16790.917} C_VEL
LIN {X 0,Y 308.132,Z 109.394,A -85,B 0,C 180,E1 -16792.308,E2 -16792.308} C_VEL
LIN {X 0,Y 310.28,Z 114.429,A -85,B 0,C 180,E1 -16792.689,E2 -16792.689} C_VEL
LIN {X 0,Y 307.954,Z 183.249,A -85,B 0,C 180,E1 -16794.311,E2 -16794.311} C_VEL
LIN {X 0,Y 307.094,Z 196.548,A -85,B 0,C 180,E1 -16794.9,E2 -16794.9} C_VEL
LIN {X 0,Y 306.028,Z 209.401,A -85,B 0,C 180,E1 -16795.766,E2 -16795.766} C_VEL
LIN {X 0,Y 304.522,Z 220.595,A -85,B 0,C 180,E1 -16796.762,E2 -16796.762} C_VEL
LIN {X 0,Y 302.585,Z 232.279,A -85,B 0,C 180,E1 -16798.102,E2 -16798.102} C_VEL
LIN {X 0,Y 300.912,Z 241.393,A -85,B 0,C 180,E1 -16799.422,E2 -16799.422} C_VEL
LIN {X 0,Y 299.164,Z 249.441,A -85,B 0,C 180,E1 -16800.826,E2 -16800.826} C_VEL
LIN {X 0,Y 297.329,Z 257.552,A -85,B 0,C 180,E1 -16802.553,E2 -16802.553} C_VEL
LIN {X 0,Y 295.419,Z 265.416,A -85,B 0,C 180,E1 -16804.645,E2 -16804.645} C_VEL
LIN {X 0,Y 293.774,Z 271.655,A -85,B 0,C 180,E1 -16806.751,E2 -16806.751} C_VEL
LIN {X 0,Y 292.47,Z 276.564,A -85,B 0,C 180,E1 -16808.872,E2 -16808.872} C_VEL
LIN {X 0,Y 291.473,Z 280.302,A -85,B 0,C 180,E1 -16811.003,E2 -16811.003} C_VEL
LIN {X 0,Y 290.648,Z 282.98,A -85,B 0,C 180,E1 -16813.132,E2 -16813.132} C_VEL
LIN {X 0,Y 290.052,Z 284.939,A -85,B 0,C 180,E1 -16815.744,E2 -16815.744} C_VEL
LIN {X 0,Y 289.791,Z 285.443,A -85,B 0,C 180,E1 -16817.393,E2 -16817.393} C_VEL
LIN {X 0,Y 289.558,Z 285.052,A -85,B 0,C 180,E1 -16820.218,E2 -16820.218} C_VEL
LIN {X 0,Y 289.632,Z 284.256,A -85,B 0,C 180,E1 -16821.628,E2 -16821.628} C_VEL
LIN {X 0,Y 289.911,Z 282.341,A -85,B 0,C 180,E1 -16823.678,E2 -16823.678} C_VEL
LIN {X 0,Y 290.039,Z 279.359,A -85,B 0,C 180,E1 -16825.831,E2 -16825.831} C_VEL
LIN {X 0,Y 290.492,Z 275.403,A -85,B 0,C 180,E1 -16827.92,E2 -16827.92} C_VEL
LIN {X 0,Y 291.082,Z 269.341,A -85,B 0,C 180,E1 -16830.346,E2 -16830.346} C_VEL
LIN {X 0,Y 292.063,Z 262.697,A -85,B 0,C 180,E1 -16832.414,E2 -16832.414} C_VEL
LIN {X 0,Y 293.103,Z 254.487,A -85,B 0,C 180,E1 -16834.47,E2 -16834.47} C_VEL
LIN {X 0,Y 294.149,Z 246.07,A -85,B 0,C 180,E1 -16836.172,E2 -16836.172} C_VEL
LIN {X 0,Y 295.572,Z 236.775,A -85,B 0,C 180,E1 -16837.686,E2 -16837.686} C_VEL
LIN {X 0,Y 296.911,Z 225.296,A -85,B 0,C 180,E1 -16839.194,E2 -16839.194} C_VEL
LIN {X 0,Y 298.018,Z 214.006,A -85,B 0,C 180,E1 -16840.359,E2 -16840.359} C_VEL
LIN {X 0,Y 298.852,Z 202.446,A -85,B 0,C 180,E1 -16841.273,E2 -16841.273} C_VEL
LIN {X 0,Y 299.537,Z 189.17,A -85,B 0,C 180,E1 -16842.019,E2 -16842.019} C_VEL
LIN {X 0,Y 299.996,Z 176.066,A -85,B 0,C 180,E1 -16842.474,E2 -16842.474} C_VEL
LIN {X 0,Y 301.49,Z 103.546,A -85,B 0,C 180,E1 -16844.187,E2 -16844.187} C_VEL
LIN {X 0,Y 294.886,Z 84.527,A -85,B 0,C 180,E1 -16845.165,E2 -16845.165} C_VEL
LIN {X 0,Y 291.579,Z 76.561,A -85,B 0,C 180,E1 -16845.632,E2 -16845.632} C_VEL
LIN {X 0,Y 291.521,Z 76.172,A -85,B 0,C 180,E1 -16845.684,E2 -16845.684} C_VEL
LIN {X 0,Y 291.452,Z 76.18,A -85,B 0,C 180,E1 -16849.875,E2 -16849.875} C_VEL
LIN {X 0,Y 291.384,Z 76.19,A -85,B 0,C 180,E1 -16854.207,E2 -16854.207} C_VEL
LIN {X 0,Y 291.422,Z 76.183,A -85,B 0,C 180,E1 -16857.272,E2 -16857.272} C_VEL
LIN {X 0,Y 291.336,Z 76.193,A -85,B 0,C 180,E1 -16860.437,E2 -16860.437} C_VEL
LIN {X 0,Y 291.346,Z 76.195,A -85,B 0,C 180,E1 -16863.699,E2 -16863.699} C_VEL
LIN {X 0,Y 291.396,Z 76.186,A -85,B 0,C 180,E1 -16867.259,E2 -16867.259} C_VEL
LIN {X 0,Y 291.352,Z 76.19,A -85,B 0,C 180,E1 -16870.64,E2 -16870.64} C_VEL
LIN {X 0,Y 291.291,Z 76.197,A -85,B 0,C 180,E1 -16874.402,E2 -16874.402} C_VEL
LIN {X 0,Y 291.328,Z 76.193,A -85,B 0,C 180,E1 -16878.405,E2 -16878.405} C_VEL
LIN {X 0,Y 291.355,Z 76.192,A -85,B 0,C 180,E1 -16881.159,E2 -16881.159} C_VEL
LIN {X 0,Y 291.363,Z 76.188,A -85,B 0,C 180,E1 -16884.627,E2 -16884.627} C_VEL
LIN {X 0,Y 291.373,Z 76.187,A -85,B 0,C 180,E1 -16887.951,E2 -16887.951} C_VEL
LIN {X 0,Y 291.377,Z 76.189,A -85,B 0,C 180,E1 -16890.993,E2 -16890.993} C_VEL
LIN {X 0,Y 290.741,Z 76.275,A -85,B 0,C 180,E1 -16892.147,E2 -16892.147} C_VEL
LIN {X 0,Y 287.927,Z 76.629,A -85,B 0,C 180,E1 -16894.026,E2 -16894.026} C_VEL
LIN {X 0,Y 285.506,Z 76.926,A -85,B 0,C 180,E1 -16895.552,E2 -16895.552} C_VEL
LIN {X 0,Y 284.44,Z 77.055,A -85,B 0,C 180,E1 -16896.734,E2 -16896.734} C_VEL
LIN {X 0,Y 284.339,Z 77.065,A -85,B 0,C 180,E1 -16897.134,E2 -16897.134} C_VEL
LIN {X 0,Y 284.407,Z 77.051,A -85,B 0,C 180,E1 -16901.262,E2 -16901.262} C_VEL
LIN {X 0,Y 284.495,Z 77.037,A -85,B 0,C 180,E1 -16904.46,E2 -16904.46} C_VEL
LIN {X 0,Y 284.487,Z 77.048,A -85,B 0,C 180,E1 -16908.602,E2 -16908.602} C_VEL
LIN {X 0,Y 284.636,Z 77.027,A -85,B 0,C 180,E1 -16911.481,E2 -16911.481} C_VEL
LIN {X 0,Y 284.598,Z 77.023,A -85,B 0,C 180,E1 -16914.331,E2 -16914.331} C_VEL
LIN {X 0,Y 284.858,Z 76.998,A -85,B 0,C 180,E1 -16918.586,E2 -16918.586} C_VEL
LIN {X 0,Y 284.858,Z 77.001,A -85,B 0,C 180,E1 -16921.414,E2 -16921.414} C_VEL
LIN {X 0,Y 284.653,Z 77.026,A -85,B 0,C 180,E1 -16927.091,E2 -16927.091} C_VEL
LIN {X 0,Y 284.518,Z 77.041,A -85,B 0,C 180,E1 -16929.957,E2 -16929.957} C_VEL
LIN {X 0,Y 284.467,Z 77.048,A -85,B 0,C 180,E1 -16934.304,E2 -16934.304} C_VEL
LIN {X 0,Y 284.39,Z 77.06,A -85,B 0,C 180,E1 -16938.74,E2 -16938.74} C_VEL
LIN {X 0,Y 284.329,Z 77.067,A -85,B 0,C 180,E1 -16941.763,E2 -16941.763} C_VEL
LIN {X 0,Y 284.32,Z 77.07,A -85,B 0,C 180,E1 -16944.849,E2 -16944.849} C_VEL
LIN {X 0,Y 284.295,Z 77.071,A -85,B 0,C 180,E1 -16948.015,E2 -16948.015} C_VEL
LIN {X 0,Y 284.29,Z 77.073,A -85,B 0,C 180,E1 -16951.275,E2 -16951.275} C_VEL
LIN {X 0,Y 284.344,Z 77.065,A -85,B 0,C 180,E1 -16955.348,E2 -16955.348} C_VEL
LIN {X 0,Y 284.315,Z 77.07,A -85,B 0,C 180,E1 -16958.169,E2 -16958.169} C_VEL
LIN {X 0,Y 284.272,Z 77.076,A -85,B 0,C 180,E1 -16962.124,E2 -16962.124} C_VEL
LIN {X 0,Y 284.258,Z 77.078,A -85,B 0,C 180,E1 -16966.189,E2 -16966.189} C_VEL
LIN {X 0,Y 284.309,Z 77.072,A -85,B 0,C 180,E1 -16970.024,E2 -16970.024} C_VEL
LIN {X 0,Y 284.332,Z 77.067,A -85,B 0,C 180,E1 -16973.613,E2 -16973.613} C_VEL
LIN {X 0,Y 284.396,Z 77.207,A -85,B 0,C 180,E1 -16976.336,E2 -16976.336} C_VEL
LIN {X 0,Y 287.125,Z 89.951,A -85,B 0,C 180,E1 -16980.286,E2 -16980.286} C_VEL
LIN {X 0,Y 288.498,Z 97.168,A -85,B 0,C 180,E1 -16982.428,E2 -16982.428} C_VEL
LIN {X 0,Y 287.96,Z 103.057,A -85,B 0,C 180,E1 -16984.029,E2 -16984.029} C_VEL
LIN {X 0,Y 292.059,Z 134.647,A -85,B 0,C 180,E1 -16985.17,E2 -16985.17} C_VEL
LIN {X 0,Y 293.985,Z 151.822,A -85,B 0,C 180,E1 -16985.752,E2 -16985.752} C_VEL
LIN {X 0,Y 292.594,Z 212.352,A -85,B 0,C 180,E1 -16987.242,E2 -16987.242} C_VEL
LIN {X 0,Y 291.786,Z 225.849,A -85,B 0,C 180,E1 -16987.846,E2 -16987.846} C_VEL
LIN {X 0,Y 290.719,Z 237.93,A -85,B 0,C 180,E1 -16988.646,E2 -16988.646} C_VEL
LIN {X 0,Y 289.379,Z 250.13,A -85,B 0,C 180,E1 -16989.752,E2 -16989.752} C_VEL
LIN {X 0,Y 287.843,Z 261.726,A -85,B 0,C 180,E1 -16991.124,E2 -16991.124} C_VEL
LIN {X 0,Y 286.521,Z 272.199,A -85,B 0,C 180,E1 -16992.698,E2 -16992.698} C_VEL
LIN {X 0,Y 285.426,Z 280.751,A -85,B 0,C 180,E1 -16994.285,E2 -16994.285} C_VEL
LIN {X 0,Y 284.249,Z 290.003,A -85,B 0,C 180,E1 -16996.415,E2 -16996.415} C_VEL
LIN {X 0,Y 283.274,Z 297.435,A -85,B 0,C 180,E1 -16998.552,E2 -16998.552} C_VEL
LIN {X 0,Y 282.821,Z 303.406,A -85,B 0,C 180,E1 -17000.705,E2 -17000.705} C_VEL
LIN {X 0,Y 282.49,Z 308.091,A -85,B 0,C 180,E1 -17002.854,E2 -17002.854} C_VEL
LIN {X 0,Y 282.485,Z 310.692,A -85,B 0,C 180,E1 -17004.368,E2 -17004.368} C_VEL
LIN {X 0,Y 282.513,Z 312.588,A -85,B 0,C 180,E1 -17005.72,E2 -17005.72} C_VEL
LIN {X 0,Y 282.534,Z 314.175,A -85,B 0,C 180,E1 -17007.148,E2 -17007.148} C_VEL
LIN {X 0,Y 282.575,Z 315.335,A -85,B 0,C 180,E1 -17008.575,E2 -17008.575} C_VEL
LIN {X 0,Y 282.661,Z 316.05,A -85,B 0,C 180,E1 -17010,E2 -17010} C_VEL
LIN {X 0,Y 282.469,Z 316.283,A -85,B 0,C 180,E1 -17012.852,E2 -17012.852} C_VEL
LIN {X 0,Y 282.392,Z 315.125,A -85,B 0,C 180,E1 -17015.437,E2 -17015.437} C_VEL
LIN {X 0,Y 282.493,Z 313.605,A -85,B 0,C 180,E1 -17017.146,E2 -17017.146} C_VEL
LIN {X 0,Y 282.871,Z 310.885,A -85,B 0,C 180,E1 -17019.294,E2 -17019.294} C_VEL
LIN {X 0,Y 283.483,Z 307.164,A -85,B 0,C 180,E1 -17021.439,E2 -17021.439} C_VEL
LIN {X 0,Y 284.616,Z 302.355,A -85,B 0,C 180,E1 -17023.567,E2 -17023.567} C_VEL
LIN {X 0,Y 286.084,Z 296.311,A -85,B 0,C 180,E1 -17025.678,E2 -17025.678} C_VEL
LIN {X 0,Y 287.87,Z 288.713,A -85,B 0,C 180,E1 -17027.798,E2 -17027.798} C_VEL
LIN {X 0,Y 289.633,Z 281.21,A -85,B 0,C 180,E1 -17029.49,E2 -17029.49} C_VEL
LIN {X 0,Y 291.825,Z 272.02,A -85,B 0,C 180,E1 -17031.177,E2 -17031.177} C_VEL
LIN {X 0,Y 294.069,Z 261.826,A -85,B 0,C 180,E1 -17032.667,E2 -17032.667} C_VEL
LIN {X 0,Y 295.955,Z 252.127,A -85,B 0,C 180,E1 -17033.81,E2 -17033.81} C_VEL
LIN {X 0,Y 298.022,Z 239.864,A -85,B 0,C 180,E1 -17034.931,E2 -17034.931} C_VEL
LIN {X 0,Y 299.751,Z 226.926,A -85,B 0,C 180,E1 -17035.799,E2 -17035.799} C_VEL
LIN {X 0,Y 300.864,Z 213.877,A -85,B 0,C 180,E1 -17036.394,E2 -17036.394} C_VEL
LIN {X 0,Y 301.702,Z 196.048,A -85,B 0,C 180,E1 -17036.86,E2 -17036.86} C_VEL
LIN {X 0,Y 302.866,Z 153.918,A -85,B 0,C 180,E1 -17037.877,E2 -17037.877} C_VEL
LIN {X 0,Y 299.52,Z 132.801,A -85,B 0,C 180,E1 -17038.856,E2 -17038.856} C_VEL
LIN {X 0,Y 295.558,Z 113.231,A -85,B 0,C 180,E1 -17039.902,E2 -17039.902} C_VEL
LIN {X 0,Y 290.388,Z 101.758,A -85,B 0,C 180,E1 -17040.938,E2 -17040.938} C_VEL
LIN {X 0,Y 288.346,Z 92.502,A -85,B 0,C 180,E1 -17044.097,E2 -17044.097} C_VEL
LIN {X 0,Y 286.386,Z 84.601,A -85,B 0,C 180,E1 -17046.958,E2 -17046.958} C_VEL
LIN {X 0,Y 284.315,Z 77.055,A -85,B 0,C 180,E1 -17049.926,E2 -17049.926} C_VEL
LIN {X 0,Y 284.247,Z 77.071,A -85,B 0,C 180,E1 -17054.19,E2 -17054.19} C_VEL
LIN {X 0,Y 284.274,Z 77.068,A -85,B 0,C 180,E1 -17058.124,E2 -17058.124} C_VEL
LIN {X 0,Y 284.325,Z 77.062,A -85,B 0,C 180,E1 -17062.278,E2 -17062.278} C_VEL
LIN {X 0,Y 284.311,Z 77.066,A -85,B 0,C 180,E1 -17065.351,E2 -17065.351} C_VEL
LIN {X 0,Y 284.299,Z 77.073,A -85,B 0,C 180,E1 -17068.726,E2 -17068.726} C_VEL
LIN {X 0,Y 284.4,Z 77.057,A -85,B 0,C 180,E1 -17072.826,E2 -17072.826} C_VEL
LIN {X 0,Y 284.37,Z 77.062,A -85,B 0,C 180,E1 -17076.707,E2 -17076.707} C_VEL
LIN {X 0,Y 284.406,Z 77.056,A -85,B 0,C 180,E1 -17081.262,E2 -17081.262} C_VEL
LIN {X 0,Y 284.495,Z 77.043,A -85,B 0,C 180,E1 -17084.459,E2 -17084.459} C_VEL
LIN {X 0,Y 284.491,Z 77.038,A -85,B 0,C 180,E1 -17088.601,E2 -17088.601} C_VEL
LIN {X 0,Y 284.643,Z 77.028,A -85,B 0,C 180,E1 -17091.48,E2 -17091.48} C_VEL
LIN {X 0,Y 284.599,Z 77.027,A -85,B 0,C 180,E1 -17094.331,E2 -17094.331} C_VEL
LIN {X 0,Y 284.857,Z 76.989,A -85,B 0,C 180,E1 -17098.586,E2 -17098.586} C_VEL
LIN {X 0,Y 284.857,Z 77.003,A -85,B 0,C 180,E1 -17101.414,E2 -17101.414} C_VEL
LIN {X 0,Y 284.676,Z 77.025,A -85,B 0,C 180,E1 -17107.09,E2 -17107.09} C_VEL
LIN {X 0,Y 284.516,Z 77.037,A -85,B 0,C 180,E1 -17109.957,E2 -17109.957} C_VEL
LIN {X 0,Y 284.466,Z 77.039,A -85,B 0,C 180,E1 -17114.303,E2 -17114.303} C_VEL
LIN {X 0,Y 284.388,Z 77.05,A -85,B 0,C 180,E1 -17118.739,E2 -17118.739} C_VEL
LIN {X 0,Y 284.328,Z 77.065,A -85,B 0,C 180,E1 -17121.763,E2 -17121.763} C_VEL
LIN {X 0,Y 284.319,Z 77.07,A -85,B 0,C 180,E1 -17124.848,E2 -17124.848} C_VEL
LIN {X 0,Y 284.293,Z 77.068,A -85,B 0,C 180,E1 -17128.015,E2 -17128.015} C_VEL
LIN {X 0,Y 284.288,Z 77.068,A -85,B 0,C 180,E1 -17131.275,E2 -17131.275} C_VEL
LIN {X 0,Y 284.338,Z 77.067,A -85,B 0,C 180,E1 -17135.346,E2 -17135.346} C_VEL
LIN {X 0,Y 284.303,Z 77.072,A -85,B 0,C 180,E1 -17138.17,E2 -17138.17} C_VEL
LIN {X 0,Y 284.269,Z 77.065,A -85,B 0,C 180,E1 -17142.124,E2 -17142.124} C_VEL
LIN {X 0,Y 284.256,Z 77.077,A -85,B 0,C 180,E1 -17146.189,E2 -17146.189} C_VEL
LIN {X 0,Y 284.286,Z 77.119,A -85,B 0,C 180,E1 -17148.264,E2 -17148.264} C_VEL
LIN {X 0,Y 285.357,Z 80.027,A -85,B 0,C 180,E1 -17148.51,E2 -17148.51} C_VEL
LIN {X 0,Y 287.003,Z 82.466,A -85,B 0,C 180,E1 -17148.821,E2 -17148.821} C_VEL
LIN {X 0,Y 293.076,Z 93.001,A -85,B 0,C 180,E1 -17149.974,E2 -17149.974} C_VEL
LIN {X 0,Y 301.346,Z 109.865,A -85,B 0,C 180,E1 -17151.513,E2 -17151.513} C_VEL
LIN {X 0,Y 304.189,Z 116.485,A -85,B 0,C 180,E1 -17152.038,E2 -17152.038} C_VEL
LIN {X 0,Y 301.883,Z 182.636,A -85,B 0,C 180,E1 -17153.614,E2 -17153.614} C_VEL
LIN {X 0,Y 301.019,Z 195.868,A -85,B 0,C 180,E1 -17154.191,E2 -17154.191} C_VEL
LIN {X 0,Y 299.978,Z 207.979,A -85,B 0,C 180,E1 -17154.989,E2 -17154.989} C_VEL
LIN {X 0,Y 298.419,Z 219.564,A -85,B 0,C 180,E1 -17155.99,E2 -17155.99} C_VEL
LIN {X 0,Y 296.409,Z 231.525,A -85,B 0,C 180,E1 -17157.356,E2 -17157.356} C_VEL
LIN {X 0,Y 294.37,Z 242.179,A -85,B 0,C 180,E1 -17158.913,E2 -17158.913} C_VEL
LIN {X 0,Y 292.42,Z 250.853,A -85,B 0,C 180,E1 -17160.482,E2 -17160.482} C_VEL
LIN {X 0,Y 290.503,Z 258.769,A -85,B 0,C 180,E1 -17162.244,E2 -17162.244} C_VEL
LIN {X 0,Y 288.601,Z 266.153,A -85,B 0,C 180,E1 -17164.292,E2 -17164.292} C_VEL
LIN {X 0,Y 287.087,Z 271.64,A -85,B 0,C 180,E1 -17166.176,E2 -17166.176} C_VEL
LIN {X 0,Y 285.669,Z 276.636,A -85,B 0,C 180,E1 -17168.344,E2 -17168.344} C_VEL
LIN {X 0,Y 284.603,Z 280.454,A -85,B 0,C 180,E1 -17170.527,E2 -17170.527} C_VEL
LIN {X 0,Y 283.72,Z 283.209,A -85,B 0,C 180,E1 -17172.707,E2 -17172.707} C_VEL
LIN {X 0,Y 282.997,Z 285.367,A -85,B 0,C 180,E1 -17175.621,E2 -17175.621} C_VEL
LIN {X 0,Y 282.74,Z 285.815,A -85,B 0,C 180,E1 -17177.073,E2 -17177.073} C_VEL
LIN {X 0,Y 282.483,Z 285.493,A -85,B 0,C 180,E1 -17179.971,E2 -17179.971} C_VEL
LIN {X 0,Y 282.529,Z 284.749,A -85,B 0,C 180,E1 -17181.416,E2 -17181.416} C_VEL
LIN {X 0,Y 282.821,Z 282.686,A -85,B 0,C 180,E1 -17183.713,E2 -17183.713} C_VEL
LIN {X 0,Y 283.033,Z 278.796,A -85,B 0,C 180,E1 -17186.441,E2 -17186.441} C_VEL
LIN {X 0,Y 283.548,Z 274.556,A -85,B 0,C 180,E1 -17188.58,E2 -17188.58} C_VEL
LIN {X 0,Y 284.286,Z 268.153,A -85,B 0,C 180,E1 -17191.063,E2 -17191.063} C_VEL
LIN {X 0,Y 285.334,Z 261.127,A -85,B 0,C 180,E1 -17193.177,E2 -17193.177} C_VEL
LIN {X 0,Y 286.502,Z 252.379,A -85,B 0,C 180,E1 -17195.278,E2 -17195.278} C_VEL
LIN {X 0,Y 287.803,Z 242.447,A -85,B 0,C 180,E1 -17197.19,E2 -17197.19} C_VEL
LIN {X 0,Y 289.129,Z 233.512,A -85,B 0,C 180,E1 -17198.562,E2 -17198.562} C_VEL
LIN {X 0,Y 290.421,Z 222.531,A -85,B 0,C 180,E1 -17199.929,E2 -17199.929} C_VEL
LIN {X 0,Y 291.545,Z 210.274,A -85,B 0,C 180,E1 -17201.119,E2 -17201.119} C_VEL
LIN {X 0,Y 292.382,Z 198.652,A -85,B 0,C 180,E1 -17201.966,E2 -17201.966} C_VEL
LIN {X 0,Y 292.979,Z 186.309,A -85,B 0,C 180,E1 -17202.596,E2 -17202.596} C_VEL
LIN {X 0,Y 293.461,Z 169.566,A -85,B 0,C 180,E1 -17203.084,E2 -17203.084} C_VEL
LIN {X 0,Y 294.921,Z 105.233,A -85,B 0,C 180,E1 -17204.628,E2 -17204.628} C_VEL
LIN {X 0,Y 288.633,Z 87.104,A -85,B 0,C 180,E1 -17205.592,E2 -17205.592} C_VEL
LIN {X 0,Y 284.587,Z 77.662,A -85,B 0,C 180,E1 -17206.177,E2 -17206.177} C_VEL
LIN {X 0,Y 284.48,Z 77.051,A -85,B 0,C 180,E1 -17206.212,E2 -17206.212} C_VEL
LIN {X 0,Y 284.378,Z 77.059,A -85,B 0,C 180,E1 -17210.243,E2 -17210.243} C_VEL
LIN {X 0,Y 284.34,Z 77.065,A -85,B 0,C 180,E1 -17214.847,E2 -17214.847} C_VEL
LIN {X 0,Y 284.33,Z 77.069,A -85,B 0,C 180,E1 -17218.011,E2 -17218.011} C_VEL
LIN {X 0,Y 284.296,Z 77.069,A -85,B 0,C 180,E1 -17221.275,E2 -17221.275} C_VEL
LIN {X 0,Y 284.363,Z 77.063,A -85,B 0,C 180,E1 -17225.354,E2 -17225.354} C_VEL
LIN {X 0,Y 284.325,Z 77.067,A -85,B 0,C 180,E1 -17228.167,E2 -17228.167} C_VEL
LIN {X 0,Y 284.284,Z 77.071,A -85,B 0,C 180,E1 -17232.128,E2 -17232.128} C_VEL
LIN {X 0,Y 284.257,Z 77.074,A -85,B 0,C 180,E1 -17236.19,E2 -17236.19} C_VEL
LIN {X 0,Y 284.308,Z 77.066,A -85,B 0,C 180,E1 -17240.024,E2 -17240.024} C_VEL
LIN {X 0,Y 284.335,Z 77.064,A -85,B 0,C 180,E1 -17243.615,E2 -17243.615} C_VEL
LIN {X 0,Y 284.31,Z 77.071,A -85,B 0,C 180,E1 -17247.19,E2 -17247.19} C_VEL
LIN {X 0,Y 284.322,Z 77.062,A -85,B 0,C 180,E1 -17250.983,E2 -17250.983} C_VEL
LIN {X 0,Y 284.379,Z 77.059,A -85,B 0,C 180,E1 -17253.587,E2 -17253.587} C_VEL
LIN {X 0,Y 284.339,Z 77.065,A -85,B 0,C 180,E1 -17257.134,E2 -17257.134} C_VEL
LIN {X 0,Y 283.633,Z 77.155,A -85,B 0,C 180,E1 -17258.316,E2 -17258.316} C_VEL
LIN {X 0,Y 280.777,Z 77.509,A -85,B 0,C 180,E1 -17260.243,E2 -17260.243} C_VEL
LIN {X 0,Y 278.408,Z 77.798,A -85,B 0,C 180,E1 -17261.808,E2 -17261.808} C_VEL
LIN {X 0,Y 277.436,Z 77.912,A -85,B 0,C 180,E1 -17263.021,E2 -17263.021} C_VEL
LIN {X 0,Y 277.379,Z 77.918,A -85,B 0,C 180,E1 -17263.431,E2 -17263.431} C_VEL
LIN {X 0,Y 277.42,Z 77.925,A -85,B 0,C 180,E1 -17266.821,E2 -17266.821} C_VEL
LIN {X 0,Y 277.601,Z 77.903,A -85,B 0,C 180,E1 -17271.263,E2 -17271.263} C_VEL
LIN {X 0,Y 277.568,Z 77.899,A -85,B 0,C 180,E1 -17274.187,E2 -17274.187} C_VEL
LIN {X 0,Y 277.824,Z 77.874,A -85,B 0,C 180,E1 -17278.551,E2 -17278.551} C_VEL
LIN {X 0,Y 277.824,Z 77.878,A -85,B 0,C 180,E1 -17281.45,E2 -17281.45} C_VEL
LIN {X 0,Y 277.611,Z 77.905,A -85,B 0,C 180,E1 -17287.272,E2 -17287.272} C_VEL
LIN {X 0,Y 277.461,Z 77.919,A -85,B 0,C 180,E1 -17290.213,E2 -17290.213} C_VEL
LIN {X 0,Y 277.414,Z 77.927,A -85,B 0,C 180,E1 -17294.675,E2 -17294.675} C_VEL
LIN {X 0,Y 277.339,Z 77.939,A -85,B 0,C 180,E1 -17299.234,E2 -17299.234} C_VEL
LIN {X 0,Y 277.292,Z 77.942,A -85,B 0,C 180,E1 -17303.924,E2 -17303.924} C_VEL
LIN {X 0,Y 277.285,Z 77.945,A -85,B 0,C 180,E1 -17307.487,E2 -17307.487} C_VEL
LIN {X 0,Y 277.251,Z 77.951,A -85,B 0,C 180,E1 -17310.473,E2 -17310.473} C_VEL
LIN {X 0,Y 277.25,Z 77.949,A -85,B 0,C 180,E1 -17313.896,E2 -17313.896} C_VEL
LIN {X 0,Y 277.271,Z 77.945,A -85,B 0,C 180,E1 -17317.469,E2 -17317.469} C_VEL
LIN {X 0,Y 277.213,Z 77.953,A -85,B 0,C 180,E1 -17321.236,E2 -17321.236} C_VEL
LIN {X 0,Y 277.204,Z 77.954,A -85,B 0,C 180,E1 -17325.226,E2 -17325.226} C_VEL
LIN {X 0,Y 277.225,Z 77.954,A -85,B 0,C 180,E1 -17329.512,E2 -17329.512} C_VEL
LIN {X 0,Y 277.265,Z 77.948,A -85,B 0,C 180,E1 -17332.53,E2 -17332.53} C_VEL
LIN {X 0,Y 277.365,Z 78.117,A -85,B 0,C 180,E1 -17335.901,E2 -17335.901} C_VEL
LIN {X 0,Y 280.01,Z 90.537,A -85,B 0,C 180,E1 -17339.868,E2 -17339.868} C_VEL
LIN {X 0,Y 281.46,Z 97.769,A -85,B 0,C 180,E1 -17342.083,E2 -17342.083} C_VEL
LIN {X 0,Y 281.259,Z 101.964,A -85,B 0,C 180,E1 -17343.27,E2 -17343.27} C_VEL
LIN {X 0,Y 281.176,Z 102.647,A -85,B 0,C 180,E1 -17343.459,E2 -17343.459} C_VEL
LIN {X 0,Y 285.289,Z 133.936,A -85,B 0,C 180,E1 -17344.638,E2 -17344.638} C_VEL
LIN {X 0,Y 287.304,Z 153.04,A -85,B 0,C 180,E1 -17345.296,E2 -17345.296} C_VEL
LIN {X 0,Y 285.87,Z 212.547,A -85,B 0,C 180,E1 -17346.8,E2 -17346.8} C_VEL
LIN {X 0,Y 285.008,Z 226.153,A -85,B 0,C 180,E1 -17347.433,E2 -17347.433} C_VEL
LIN {X 0,Y 283.866,Z 238.589,A -85,B 0,C 180,E1 -17348.295,E2 -17348.295} C_VEL
LIN {X 0,Y 282.489,Z 250.505,A -85,B 0,C 180,E1 -17349.426,E2 -17349.426} C_VEL
LIN {X 0,Y 280.908,Z 261.962,A -85,B 0,C 180,E1 -17350.83,E2 -17350.83} C_VEL
LIN {X 0,Y 279.548,Z 272.309,A -85,B 0,C 180,E1 -17352.441,E2 -17352.441} C_VEL
LIN {X 0,Y 278.452,Z 279.886,A -85,B 0,C 180,E1 -17353.881,E2 -17353.881} C_VEL
LIN {X 0,Y 277.43,Z 287.86,A -85,B 0,C 180,E1 -17355.7,E2 -17355.7} C_VEL
LIN {X 0,Y 276.446,Z 295.624,A -85,B 0,C 180,E1 -17357.893,E2 -17357.893} C_VEL
LIN {X 0,Y 275.754,Z 302.778,A -85,B 0,C 180,E1 -17360.464,E2 -17360.464} C_VEL
LIN {X 0,Y 275.441,Z 307.519,A -85,B 0,C 180,E1 -17362.67,E2 -17362.67} C_VEL
LIN {X 0,Y 275.398,Z 310.46,A -85,B 0,C 180,E1 -17364.422,E2 -17364.422} C_VEL
LIN {X 0,Y 275.457,Z 313.696,A -85,B 0,C 180,E1 -17367.075,E2 -17367.075} C_VEL
LIN {X 0,Y 275.488,Z 314.89,A -85,B 0,C 180,E1 -17368.538,E2 -17368.538} C_VEL
LIN {X 0,Y 275.571,Z 315.634,A -85,B 0,C 180,E1 -17370,E2 -17370} C_VEL
LIN {X 0,Y 275.392,Z 315.908,A -85,B 0,C 180,E1 -17372.926,E2 -17372.926} C_VEL
LIN {X 0,Y 275.309,Z 314.909,A -85,B 0,C 180,E1 -17375.386,E2 -17375.386} C_VEL
LIN {X 0,Y 275.424,Z 313.313,A -85,B 0,C 180,E1 -17377.33,E2 -17377.33} C_VEL
LIN {X 0,Y 275.849,Z 310.637,A -85,B 0,C 180,E1 -17379.532,E2 -17379.532} C_VEL
LIN {X 0,Y 276.478,Z 306.962,A -85,B 0,C 180,E1 -17381.733,E2 -17381.733} C_VEL
LIN {X 0,Y 277.684,Z 302.206,A -85,B 0,C 180,E1 -17383.912,E2 -17383.912} C_VEL
LIN {X 0,Y 279.217,Z 296.221,A -85,B 0,C 180,E1 -17386.074,E2 -17386.074} C_VEL
LIN {X 0,Y 280.949,Z 289.28,A -85,B 0,C 180,E1 -17388.087,E2 -17388.087} C_VEL
LIN {X 0,Y 282.943,Z 281.263,A -85,B 0,C 180,E1 -17389.97,E2 -17389.97} C_VEL
LIN {X 0,Y 285.221,Z 272.169,A -85,B 0,C 180,E1 -17391.691,E2 -17391.691} C_VEL
LIN {X 0,Y 287.55,Z 262.138,A -85,B 0,C 180,E1 -17393.211,E2 -17393.211} C_VEL
LIN {X 0,Y 289.79,Z 251.021,A -85,B 0,C 180,E1 -17394.539,E2 -17394.539} C_VEL
LIN {X 0,Y 291.913,Z 238.576,A -85,B 0,C 180,E1 -17395.681,E2 -17395.681} C_VEL
LIN {X 0,Y 293.645,Z 225.919,A -85,B 0,C 180,E1 -17396.52,E2 -17396.52} C_VEL
LIN {X 0,Y 294.877,Z 212.279,A -85,B 0,C 180,E1 -17397.128,E2 -17397.128} C_VEL
LIN {X 0,Y 296.014,Z 184.109,A -85,B 0,C 180,E1 -17397.84,E2 -17397.84} C_VEL
LIN {X 0,Y 296.835,Z 154.97,A -85,B 0,C 180,E1 -17398.559,E2 -17398.559} C_VEL
LIN {X 0,Y 292.992,Z 130.774,A -85,B 0,C 180,E1 -17399.726,E2 -17399.726} C_VEL
LIN {X 0,Y 289.798,Z 115.856,A -85,B 0,C 180,E1 -17400.581,E2 -17400.581} C_VEL
LIN {X 0,Y 283.156,Z 101.254,A -85,B 0,C 180,E1 -17401.977,E2 -17401.977} C_VEL
LIN {X 0,Y 280.606,Z 90.177,A -85,B 0,C 180,E1 -17405.946,E2 -17405.946} C_VEL
LIN {X 0,Y 278.104,Z 81.023,A -85,B 0,C 180,E1 -17409.532,E2 -17409.532} C_VEL
LIN {X 0,Y 277.233,Z 77.946,A -85,B 0,C 180,E1 -17410.84,E2 -17410.84} C_VEL
LIN {X 0,Y 277.203,Z 77.947,A -85,B 0,C 180,E1 -17415.226,E2 -17415.226} C_VEL
LIN {X 0,Y 277.225,Z 77.943,A -85,B 0,C 180,E1 -17419.512,E2 -17419.512} C_VEL
LIN {X 0,Y 277.27,Z 77.939,A -85,B 0,C 180,E1 -17422.531,E2 -17422.531} C_VEL
LIN {X 0,Y 277.249,Z 77.941,A -85,B 0,C 180,E1 -17426.104,E2 -17426.104} C_VEL
LIN {X 0,Y 277.264,Z 77.941,A -85,B 0,C 180,E1 -17429.539,E2 -17429.539} C_VEL
LIN {X 0,Y 277.362,Z 77.933,A -85,B 0,C 180,E1 -17432.864,E2 -17432.864} C_VEL
LIN {X 0,Y 277.332,Z 77.939,A -85,B 0,C 180,E1 -17436.08,E2 -17436.08} C_VEL
LIN {X 0,Y 277.348,Z 77.938,A -85,B 0,C 180,E1 -17440.766,E2 -17440.766} C_VEL
LIN {X 0,Y 277.438,Z 77.925,A -85,B 0,C 180,E1 -17445.326,E2 -17445.326} C_VEL
LIN {X 0,Y 277.464,Z 77.92,A -85,B 0,C 180,E1 -17449.787,E2 -17449.787} C_VEL
LIN {X 0,Y 277.644,Z 77.886,A -85,B 0,C 180,E1 -17452.729,E2 -17452.729} C_VEL
LIN {X 0,Y 277.823,Z 77.865,A -85,B 0,C 180,E1 -17458.55,E2 -17458.55} C_VEL
LIN {X 0,Y 277.823,Z 77.88,A -85,B 0,C 180,E1 -17461.449,E2 -17461.449} C_VEL
LIN {X 0,Y 277.63,Z 77.899,A -85,B 0,C 180,E1 -17467.271,E2 -17467.271} C_VEL
LIN {X 0,Y 277.46,Z 77.919,A -85,B 0,C 180,E1 -17470.213,E2 -17470.213} C_VEL
LIN {X 0,Y 277.412,Z 77.919,A -85,B 0,C 180,E1 -17474.675,E2 -17474.675} C_VEL
LIN {X 0,Y 277.337,Z 77.93,A -85,B 0,C 180,E1 -17479.234,E2 -17479.234} C_VEL
LIN {X 0,Y 277.291,Z 77.939,A -85,B 0,C 180,E1 -17483.924,E2 -17483.924} C_VEL
LIN {X 0,Y 277.283,Z 77.939,A -85,B 0,C 180,E1 -17487.487,E2 -17487.487} C_VEL
LIN {X 0,Y 277.249,Z 77.944,A -85,B 0,C 180,E1 -17490.472,E2 -17490.472} C_VEL
LIN {X 0,Y 277.247,Z 77.945,A -85,B 0,C 180,E1 -17493.896,E2 -17493.896} C_VEL
LIN {X 0,Y 277.257,Z 77.945,A -85,B 0,C 180,E1 -17497.471,E2 -17497.471} C_VEL
LIN {X 0,Y 277.209,Z 77.936,A -85,B 0,C 180,E1 -17501.236,E2 -17501.236} C_VEL
LIN {X 0,Y 277.201,Z 77.959,A -85,B 0,C 180,E1 -17505.226,E2 -17505.226} C_VEL
LIN {X 0,Y 277.192,Z 77.96,A -85,B 0,C 180,E1 -17507.208,E2 -17507.208} C_VEL
LIN {X 0,Y 278.256,Z 80.89,A -85,B 0,C 180,E1 -17507.472,E2 -17507.472} C_VEL
LIN {X 0,Y 279.942,Z 83.24,A -85,B 0,C 180,E1 -17507.805,E2 -17507.805} C_VEL
LIN {X 0,Y 287.575,Z 96.183,A -85,B 0,C 180,E1 -17509.315,E2 -17509.315} C_VEL
LIN {X 0,Y 295.541,Z 112.434,A -85,B 0,C 180,E1 -17510.86,E2 -17510.86} C_VEL
LIN {X 0,Y 298.233,Z 118.827,A -85,B 0,C 180,E1 -17511.38,E2 -17511.38} C_VEL
LIN {X 0,Y 295.759,Z 183.474,A -85,B 0,C 180,E1 -17512.939,E2 -17512.939} C_VEL
LIN {X 0,Y 294.871,Z 196.512,A -85,B 0,C 180,E1 -17513.524,E2 -17513.524} C_VEL
LIN {X 0,Y 293.65,Z 209.696,A -85,B 0,C 180,E1 -17514.423,E2 -17514.423} C_VEL
LIN {X 0,Y 292.131,Z 220.188,A -85,B 0,C 180,E1 -17515.364,E2 -17515.364} C_VEL
LIN {X 0,Y 290.041,Z 232.095,A -85,B 0,C 180,E1 -17516.754,E2 -17516.754} C_VEL
LIN {X 0,Y 287.83,Z 243.167,A -85,B 0,C 180,E1 -17518.416,E2 -17518.416} C_VEL
LIN {X 0,Y 285.668,Z 252.209,A -85,B 0,C 180,E1 -17520.12,E2 -17520.12} C_VEL
LIN {X 0,Y 283.682,Z 259.941,A -85,B 0,C 180,E1 -17521.919,E2 -17521.919} C_VEL
LIN {X 0,Y 281.864,Z 266.667,A -85,B 0,C 180,E1 -17523.847,E2 -17523.847} C_VEL
LIN {X 0,Y 279.88,Z 273.46,A -85,B 0,C 180,E1 -17526.311,E2 -17526.311} C_VEL
LIN {X 0,Y 278.443,Z 278.287,A -85,B 0,C 180,E1 -17528.609,E2 -17528.609} C_VEL
LIN {X 0,Y 277.403,Z 281.676,A -85,B 0,C 180,E1 -17530.77,E2 -17530.77} C_VEL
LIN {X 0,Y 276.802,Z 283.438,A -85,B 0,C 180,E1 -17532.261,E2 -17532.261} C_VEL
LIN {X 0,Y 276.303,Z 284.756,A -85,B 0,C 180,E1 -17533.752,E2 -17533.752} C_VEL
LIN {X 0,Y 275.96,Z 285.754,A -85,B 0,C 180,E1 -17535.412,E2 -17535.412} C_VEL
LIN {X 0,Y 275.494,Z 286.254,A -85,B 0,C 180,E1 -17538.224,E2 -17538.224} C_VEL
LIN {X 0,Y 275.419,Z 285.226,A -85,B 0,C 180,E1 -17541.193,E2 -17541.193} C_VEL
LIN {X 0,Y 275.748,Z 283.065,A -85,B 0,C 180,E1 -17543.717,E2 -17543.717} C_VEL
LIN {X 0,Y 275.936,Z 279.452,A -85,B 0,C 180,E1 -17546.349,E2 -17546.349} C_VEL
LIN {X 0,Y 276.454,Z 275.292,A -85,B 0,C 180,E1 -17548.543,E2 -17548.543} C_VEL
LIN {X 0,Y 277.212,Z 268.975,A -85,B 0,C 180,E1 -17551.09,E2 -17551.09} C_VEL
LIN {X 0,Y 278.286,Z 262.083,A -85,B 0,C 180,E1 -17553.258,E2 -17553.258} C_VEL
LIN {X 0,Y 279.463,Z 253.47,A -85,B 0,C 180,E1 -17555.412,E2 -17555.412} C_VEL
LIN {X 0,Y 280.66,Z 244.652,A -85,B 0,C 180,E1 -17557.193,E2 -17557.193} C_VEL
LIN {X 0,Y 282.181,Z 234.915,A -85,B 0,C 180,E1 -17558.775,E2 -17558.775} C_VEL
LIN {X 0,Y 283.499,Z 224.266,A -85,B 0,C 180,E1 -17560.174,E2 -17560.174} C_VEL
LIN {X 0,Y 284.68,Z 212.355,A -85,B 0,C 180,E1 -17561.391,E2 -17561.391} C_VEL
LIN {X 0,Y 285.571,Z 199.989,A -85,B 0,C 180,E1 -17562.345,E2 -17562.345} C_VEL
LIN {X 0,Y 286.277,Z 187.093,A -85,B 0,C 180,E1 -17563.035,E2 -17563.035} C_VEL
LIN {X 0,Y 286.753,Z 171.599,A -85,B 0,C 180,E1 -17563.509,E2 -17563.509} C_VEL
LIN {X 0,Y 288.199,Z 106.331,A -85,B 0,C 180,E1 -17565.118,E2 -17565.118} C_VEL
LIN {X 0,Y 282.253,Z 89.396,A -85,B 0,C 180,E1 -17566.057,E2 -17566.057} C_VEL
LIN {X 0,Y 277.576,Z 78.772,A -85,B 0,C 180,E1 -17566.752,E2 -17566.752} C_VEL
LIN {X 0,Y 277.401,Z 77.931,A -85,B 0,C 180,E1 -17566.845,E2 -17566.845} C_VEL
LIN {X 0,Y 277.292,Z 77.94,A -85,B 0,C 180,E1 -17570.783,E2 -17570.783} C_VEL
LIN {X 0,Y 277.293,Z 77.945,A -85,B 0,C 180,E1 -17574.158,E2 -17574.158} C_VEL
LIN {X 0,Y 277.326,Z 77.939,A -85,B 0,C 180,E1 -17577.505,E2 -17577.505} C_VEL
LIN {X 0,Y 277.273,Z 77.945,A -85,B 0,C 180,E1 -17580.482,E2 -17580.482} C_VEL
LIN {X 0,Y 277.256,Z 77.949,A -85,B 0,C 180,E1 -17583.895,E2 -17583.895} C_VEL
LIN {X 0,Y 277.283,Z 77.945,A -85,B 0,C 180,E1 -17587.467,E2 -17587.467} C_VEL
LIN {X 0,Y 277.223,Z 77.952,A -85,B 0,C 180,E1 -17591.235,E2 -17591.235} C_VEL
LIN {X 0,Y 277.202,Z 77.954,A -85,B 0,C 180,E1 -17595.227,E2 -17595.227} C_VEL
LIN {X 0,Y 277.225,Z 77.951,A -85,B 0,C 180,E1 -17599.512,E2 -17599.512} C_VEL
LIN {X 0,Y 277.27,Z 77.945,A -85,B 0,C 180,E1 -17602.531,E2 -17602.531} C_VEL
LIN {X 0,Y 277.249,Z 77.946,A -85,B 0,C 180,E1 -17606.105,E2 -17606.105} C_VEL
LIN {X 0,Y 277.264,Z 77.944,A -85,B 0,C 180,E1 -17609.539,E2 -17609.539} C_VEL
LIN {X 0,Y 277.36,Z 77.937,A -85,B 0,C 180,E1 -17612.864,E2 -17612.864} C_VEL
LIN {X 0,Y 277.28,Z 77.94,A -85,B 0,C 180,E1 -17617.132,E2 -17617.132} C_VEL
LIN {X 0,Y 277.348,Z 77.932,A -85,B 0,C 180,E1 -17620.767,E2 -17620.767} C_VEL
LIN {X 0,Y 277.379,Z 77.918,A -85,B 0,C 180,E1 -17623.431,E2 -17623.431} C_VEL
LIN {X 0,Y 276.762,Z 78,A -85,B 0,C 180,E1 -17624.643,E2 -17624.643} C_VEL
LIN {X 0,Y 273.913,Z 78.363,A -85,B 0,C 180,E1 -17626.617,E2 -17626.617} C_VEL
LIN {X 0,Y 271.49,Z 78.667,A -85,B 0,C 180,E1 -17628.221,E2 -17628.221} C_VEL
LIN {X 0,Y 270.49,Z 78.79,A -85,B 0,C 180,E1 -17629.465,E2 -17629.465} C_VEL
LIN {X 0,Y 270.432,Z 78.795,A -85,B 0,C 180,E1 -17629.887,E2 -17629.887} C_VEL
LIN {X 0,Y 270.599,Z 78.772,A -85,B 0,C 180,E1 -17632.539,E2 -17632.539} C_VEL
LIN {X 0,Y 270.79,Z 78.75,A -85,B 0,C 180,E1 -17638.513,E2 -17638.513} C_VEL
LIN {X 0,Y 270.79,Z 78.754,A -85,B 0,C 180,E1 -17641.487,E2 -17641.487} C_VEL
LIN {X 0,Y 270.571,Z 78.783,A -85,B 0,C 180,E1 -17647.462,E2 -17647.462} C_VEL
LIN {X 0,Y 270.414,Z 78.796,A -85,B 0,C 180,E1 -17650.482,E2 -17650.482} C_VEL
LIN {X 0,Y 270.381,Z 78.805,A -85,B 0,C 180,E1 -17655.066,E2 -17655.066} C_VEL
LIN {X 0,Y 270.301,Z 78.812,A -85,B 0,C 180,E1 -17659.756,E2 -17659.756} C_VEL
LIN {X 0,Y 270.234,Z 78.823,A -85,B 0,C 180,E1 -17664.59,E2 -17664.59} C_VEL
LIN {X 0,Y 270.212,Z 78.825,A -85,B 0,C 180,E1 -17667.916,E2 -17667.916} C_VEL
LIN {X 0,Y 270.177,Z 78.831,A -85,B 0,C 180,E1 -17671.349,E2 -17671.349} C_VEL
LIN {X 0,Y 270.205,Z 78.828,A -85,B 0,C 180,E1 -17674.905,E2 -17674.905} C_VEL
LIN {X 0,Y 270.2,Z 78.828,A -85,B 0,C 180,E1 -17678.71,E2 -17678.71} C_VEL
LIN {X 0,Y 270.175,Z 78.83,A -85,B 0,C 180,E1 -17682.558,E2 -17682.558} C_VEL
LIN {X 0,Y 270.168,Z 78.832,A -85,B 0,C 180,E1 -17686.751,E2 -17686.751} C_VEL
LIN {X 0,Y 270.2,Z 78.828,A -85,B 0,C 180,E1 -17691.289,E2 -17691.289} C_VEL
LIN {X 0,Y 270.282,Z 78.928,A -85,B 0,C 180,E1 -17695.414,E2 -17695.414} C_VEL
LIN {X 0,Y 272.903,Z 91.113,A -85,B 0,C 180,E1 -17699.428,E2 -17699.428} C_VEL
LIN {X 0,Y 274.57,Z 99.791,A -85,B 0,C 180,E1 -17702.151,E2 -17702.151} C_VEL
LIN {X 0,Y 274.397,Z 102.294,A -85,B 0,C 180,E1 -17702.874,E2 -17702.874} C_VEL
LIN {X 0,Y 278.531,Z 133.222,A -85,B 0,C 180,E1 -17704.08,E2 -17704.08} C_VEL
LIN {X 0,Y 280.657,Z 153.643,A -85,B 0,C 180,E1 -17704.805,E2 -17704.805} C_VEL
LIN {X 0,Y 279.209,Z 211.673,A -85,B 0,C 180,E1 -17706.3,E2 -17706.3} C_VEL
LIN {X 0,Y 278.371,Z 224.867,A -85,B 0,C 180,E1 -17706.913,E2 -17706.913} C_VEL
LIN {X 0,Y 277.202,Z 236.998,A -85,B 0,C 180,E1 -17707.745,E2 -17707.745} C_VEL
LIN {X 0,Y 275.803,Z 249.256,A -85,B 0,C 180,E1 -17708.904,E2 -17708.904} C_VEL
LIN {X 0,Y 274.209,Z 260.881,A -85,B 0,C 180,E1 -17710.342,E2 -17710.342} C_VEL
LIN {X 0,Y 272.764,Z 271.367,A -85,B 0,C 180,E1 -17711.989,E2 -17711.989} C_VEL
LIN {X 0,Y 271.391,Z 280.768,A -85,B 0,C 180,E1 -17713.836,E2 -17713.836} C_VEL
LIN {X 0,Y 270.167,Z 289.883,A -85,B 0,C 180,E1 -17716.076,E2 -17716.076} C_VEL
LIN {X 0,Y 269.144,Z 297.203,A -85,B 0,C 180,E1 -17718.324,E2 -17718.324} C_VEL
LIN {X 0,Y 268.693,Z 302.151,A -85,B 0,C 180,E1 -17720.211,E2 -17720.211} C_VEL
LIN {X 0,Y 268.362,Z 306.945,A -85,B 0,C 180,E1 -17722.476,E2 -17722.476} C_VEL
LIN {X 0,Y 268.32,Z 310.196,A -85,B 0,C 180,E1 -17724.457,E2 -17724.457} C_VEL
LIN {X 0,Y 268.383,Z 313.217,A -85,B 0,C 180,E1 -17726.998,E2 -17726.998} C_VEL
LIN {X 0,Y 268.404,Z 314.436,A -85,B 0,C 180,E1 -17728.499,E2 -17728.499} C_VEL
LIN {X 0,Y 268.481,Z 315.218,A -85,B 0,C 180,E1 -17730,E2 -17730} C_VEL
LIN {X 0,Y 268.316,Z 315.534,A -85,B 0,C 180,E1 -17733.003,E2 -17733.003} C_VEL
LIN {X 0,Y 268.241,Z 314.667,A -85,B 0,C 180,E1 -17735.366,E2 -17735.366} C_VEL
LIN {X 0,Y 268.345,Z 313.022,A -85,B 0,C 180,E1 -17737.524,E2 -17737.524} C_VEL
LIN {X 0,Y 268.795,Z 310.392,A -85,B 0,C 180,E1 -17739.785,E2 -17739.785} C_VEL
LIN {X 0,Y 269.487,Z 306.767,A -85,B 0,C 180,E1 -17742.042,E2 -17742.042} C_VEL
LIN {X 0,Y 270.773,Z 302.064,A -85,B 0,C 180,E1 -17744.275,E2 -17744.275} C_VEL
LIN {X 0,Y 272.7,Z 295.015,A -85,B 0,C 180,E1 -17746.854,E2 -17746.854} C_VEL
LIN {X 0,Y 274.67,Z 287.43,A -85,B 0,C 180,E1 -17749.037,E2 -17749.037} C_VEL
LIN {X 0,Y 276.714,Z 279.687,A -85,B 0,C 180,E1 -17750.829,E2 -17750.829} C_VEL
LIN {X 0,Y 279.393,Z 269.217,A -85,B 0,C 180,E1 -17752.752,E2 -17752.752} C_VEL
LIN {X 0,Y 281.839,Z 258.59,A -85,B 0,C 180,E1 -17754.296,E2 -17754.296} C_VEL
LIN {X 0,Y 284.004,Z 248.335,A -85,B 0,C 180,E1 -17755.465,E2 -17755.465} C_VEL
LIN {X 0,Y 286.081,Z 236.16,A -85,B 0,C 180,E1 -17756.539,E2 -17756.539} C_VEL
LIN {X 0,Y 287.859,Z 222.637,A -85,B 0,C 180,E1 -17757.391,E2 -17757.391} C_VEL
LIN {X 0,Y 288.925,Z 210.157,A -85,B 0,C 180,E1 -17757.917,E2 -17757.917} C_VEL
LIN {X 0,Y 290.823,Z 156.072,A -85,B 0,C 180,E1 -17759.272,E2 -17759.272} C_VEL
LIN {X 0,Y 287.122,Z 132.441,A -85,B 0,C 180,E1 -17760.45,E2 -17760.45} C_VEL
LIN {X 0,Y 284.282,Z 118.894,A -85,B 0,C 180,E1 -17761.247,E2 -17761.247} C_VEL
LIN {X 0,Y 277.263,Z 104.036,A -85,B 0,C 180,E1 -17762.733,E2 -17762.733} C_VEL
LIN {X 0,Y 275.844,Z 100.766,A -85,B 0,C 180,E1 -17763.083,E2 -17763.083} C_VEL
LIN {X 0,Y 273.305,Z 89.966,A -85,B 0,C 180,E1 -17767.14,E2 -17767.14} C_VEL
LIN {X 0,Y 271.066,Z 82.017,A -85,B 0,C 180,E1 -17770.405,E2 -17770.405} C_VEL
LIN {X 0,Y 270.163,Z 78.828,A -85,B 0,C 180,E1 -17771.859,E2 -17771.859} C_VEL
LIN {X 0,Y 270.154,Z 78.826,A -85,B 0,C 180,E1 -17775.38,E2 -17775.38} C_VEL
LIN {X 0,Y 270.176,Z 78.821,A -85,B 0,C 180,E1 -17779.434,E2 -17779.434} C_VEL
LIN {X 0,Y 270.228,Z 78.815,A -85,B 0,C 180,E1 -17783.73,E2 -17783.73} C_VEL
LIN {X 0,Y 270.205,Z 78.818,A -85,B 0,C 180,E1 -17786.893,E2 -17786.893} C_VEL
LIN {X 0,Y 270.231,Z 78.815,A -85,B 0,C 180,E1 -17790.387,E2 -17790.387} C_VEL
LIN {X 0,Y 270.267,Z 78.81,A -85,B 0,C 180,E1 -17793.764,E2 -17793.764} C_VEL
LIN {X 0,Y 270.236,Z 78.819,A -85,B 0,C 180,E1 -17797.039,E2 -17797.039} C_VEL
LIN {X 0,Y 270.304,Z 78.813,A -85,B 0,C 180,E1 -17800.244,E2 -17800.244} C_VEL
LIN {X 0,Y 270.406,Z 78.803,A -85,B 0,C 180,E1 -17804.935,E2 -17804.935} C_VEL
LIN {X 0,Y 270.416,Z 78.797,A -85,B 0,C 180,E1 -17809.518,E2 -17809.518} C_VEL
LIN {X 0,Y 270.602,Z 78.764,A -85,B 0,C 180,E1 -17812.538,E2 -17812.538} C_VEL
LIN {X 0,Y 270.789,Z 78.741,A -85,B 0,C 180,E1 -17818.513,E2 -17818.513} C_VEL
LIN {X 0,Y 270.789,Z 78.756,A -85,B 0,C 180,E1 -17821.487,E2 -17821.487} C_VEL
LIN {X 0,Y 270.587,Z 78.774,A -85,B 0,C 180,E1 -17827.462,E2 -17827.462} C_VEL
LIN {X 0,Y 270.412,Z 78.798,A -85,B 0,C 180,E1 -17830.482,E2 -17830.482} C_VEL
LIN {X 0,Y 270.38,Z 78.798,A -85,B 0,C 180,E1 -17835.066,E2 -17835.066} C_VEL
LIN {X 0,Y 270.299,Z 78.811,A -85,B 0,C 180,E1 -17839.756,E2 -17839.756} C_VEL
LIN {X 0,Y 270.232,Z 78.822,A -85,B 0,C 180,E1 -17844.589,E2 -17844.589} C_VEL
LIN {X 0,Y 270.21,Z 78.822,A -85,B 0,C 180,E1 -17847.915,E2 -17847.915} C_VEL
LIN {X 0,Y 270.175,Z 78.826,A -85,B 0,C 180,E1 -17851.349,E2 -17851.349} C_VEL
LIN {X 0,Y 270.199,Z 78.826,A -85,B 0,C 180,E1 -17854.906,E2 -17854.906} C_VEL
LIN {X 0,Y 270.198,Z 78.829,A -85,B 0,C 180,E1 -17858.71,E2 -17858.71} C_VEL
LIN {X 0,Y 270.172,Z 78.826,A -85,B 0,C 180,E1 -17862.558,E2 -17862.558} C_VEL
LIN {X 0,Y 270.148,Z 78.862,A -85,B 0,C 180,E1 -17866.096,E2 -17866.096} C_VEL
LIN {X 0,Y 271.117,Z 81.639,A -85,B 0,C 180,E1 -17866.35,E2 -17866.35} C_VEL
LIN {X 0,Y 272.883,Z 84.071,A -85,B 0,C 180,E1 -17866.72,E2 -17866.72} C_VEL
LIN {X 0,Y 281.038,Z 97.444,A -85,B 0,C 180,E1 -17868.413,E2 -17868.413} C_VEL
LIN {X 0,Y 288.774,Z 112.885,A -85,B 0,C 180,E1 -17869.979,E2 -17869.979} C_VEL
LIN {X 0,Y 292.19,Z 120.615,A -85,B 0,C 180,E1 -17870.661,E2 -17870.661} C_VEL
LIN {X 0,Y 289.657,Z 184.511,A -85,B 0,C 180,E1 -17872.241,E2 -17872.241} C_VEL
LIN {X 0,Y 288.734,Z 197.47,A -85,B 0,C 180,E1 -17872.846,E2 -17872.846} C_VEL
LIN {X 0,Y 287.545,Z 209.662,A -85,B 0,C 180,E1 -17873.695,E2 -17873.695} C_VEL
LIN {X 0,Y 285.892,Z 220.809,A -85,B 0,C 180,E1 -17874.711,E2 -17874.711} C_VEL
LIN {X 0,Y 283.705,Z 232.665,A -85,B 0,C 180,E1 -17876.125,E2 -17876.125} C_VEL
LIN {X 0,Y 281.515,Z 243.275,A -85,B 0,C 180,E1 -17877.749,E2 -17877.749} C_VEL
LIN {X 0,Y 279.311,Z 252.076,A -85,B 0,C 180,E1 -17879.417,E2 -17879.417} C_VEL
LIN {X 0,Y 276.886,Z 261.111,A -85,B 0,C 180,E1 -17881.581,E2 -17881.581} C_VEL
LIN {X 0,Y 274.932,Z 267.896,A -85,B 0,C 180,E1 -17883.617,E2 -17883.617} C_VEL
LIN {X 0,Y 273.21,Z 273.454,A -85,B 0,C 180,E1 -17885.696,E2 -17885.696} C_VEL
LIN {X 0,Y 271.701,Z 278.224,A -85,B 0,C 180,E1 -17887.971,E2 -17887.971} C_VEL
LIN {X 0,Y 270.545,Z 281.834,A -85,B 0,C 180,E1 -17890.263,E2 -17890.263} C_VEL
LIN {X 0,Y 269.878,Z 283.669,A -85,B 0,C 180,E1 -17891.79,E2 -17891.79} C_VEL
LIN {X 0,Y 269.337,Z 285.024,A -85,B 0,C 180,E1 -17893.32,E2 -17893.32} C_VEL
LIN {X 0,Y 268.916,Z 286.164,A -85,B 0,C 180,E1 -17895.235,E2 -17895.235} C_VEL
LIN {X 0,Y 268.46,Z 286.66,A -85,B 0,C 180,E1 -17897.911,E2 -17897.911} C_VEL
LIN {X 0,Y 268.329,Z 285.701,A -85,B 0,C 180,E1 -17900.959,E2 -17900.959} C_VEL
LIN {X 0,Y 268.67,Z 283.429,A -85,B 0,C 180,E1 -17903.731,E2 -17903.731} C_VEL
LIN {X 0,Y 268.843,Z 280.103,A -85,B 0,C 180,E1 -17906.253,E2 -17906.253} C_VEL
LIN {X 0,Y 269.362,Z 276.022,A -85,B 0,C 180,E1 -17908.505,E2 -17908.505} C_VEL
LIN {X 0,Y 270.141,Z 269.788,A -85,B 0,C 180,E1 -17911.118,E2 -17911.118} C_VEL
LIN {X 0,Y 271.206,Z 262.996,A -85,B 0,C 180,E1 -17913.343,E2 -17913.343} C_VEL
LIN {X 0,Y 272.43,Z 254.546,A -85,B 0,C 180,E1 -17915.552,E2 -17915.552} C_VEL
LIN {X 0,Y 273.654,Z 245.867,A -85,B 0,C 180,E1 -17917.378,E2 -17917.378} C_VEL
LIN {X 0,Y 275.221,Z 236.296,A -85,B 0,C 180,E1 -17918.999,E2 -17918.999} C_VEL
LIN {X 0,Y 276.584,Z 225.877,A -85,B 0,C 180,E1 -17920.431,E2 -17920.431} C_VEL
LIN {X 0,Y 277.816,Z 214.416,A -85,B 0,C 180,E1 -17921.676,E2 -17921.676} C_VEL
LIN {X 0,Y 278.752,Z 202.566,A -85,B 0,C 180,E1 -17922.652,E2 -17922.652} C_VEL
LIN {X 0,Y 279.49,Z 189.774,A -85,B 0,C 180,E1 -17923.404,E2 -17923.404} C_VEL
LIN {X 0,Y 279.988,Z 176.268,A -85,B 0,C 180,E1 -17923.888,E2 -17923.888} C_VEL
LIN {X 0,Y 281.587,Z 107.754,A -85,B 0,C 180,E1 -17925.614,E2 -17925.614} C_VEL
LIN {X 0,Y 275.786,Z 91.431,A -85,B 0,C 180,E1 -17926.558,E2 -17926.558} C_VEL
LIN {X 0,Y 270.428,Z 79.362,A -85,B 0,C 180,E1 -17927.386,E2 -17927.386} C_VEL
LIN {X 0,Y 270.338,Z 78.81,A -85,B 0,C 180,E1 -17927.434,E2 -17927.434} C_VEL
LIN {X 0,Y 270.215,Z 78.821,A -85,B 0,C 180,E1 -17931.354,E2 -17931.354} C_VEL
LIN {X 0,Y 270.239,Z 78.823,A -85,B 0,C 180,E1 -17934.589,E2 -17934.589} C_VEL
LIN {X 0,Y 270.271,Z 78.82,A -85,B 0,C 180,E1 -17937.909,E2 -17937.909} C_VEL
LIN {X 0,Y 270.185,Z 78.827,A -85,B 0,C 180,E1 -17941.348,E2 -17941.348} C_VEL
LIN {X 0,Y 270.225,Z 78.822,A -85,B 0,C 180,E1 -17944.903,E2 -17944.903} C_VEL
LIN {X 0,Y 270.224,Z 78.823,A -85,B 0,C 180,E1 -17948.717,E2 -17948.717} C_VEL
LIN {X 0,Y 270.17,Z 78.831,A -85,B 0,C 180,E1 -17953.25,E2 -17953.25} C_VEL
LIN {X 0,Y 270.173,Z 78.832,A -85,B 0,C 180,E1 -17957.442,E2 -17957.442} C_VEL
LIN {X 0,Y 270.209,Z 78.827,A -85,B 0,C 180,E1 -17961.375,E2 -17961.375} C_VEL
LIN {X 0,Y 270.204,Z 78.825,A -85,B 0,C 180,E1 -17965.095,E2 -17965.095} C_VEL
LIN {X 0,Y 270.203,Z 78.825,A -85,B 0,C 180,E1 -17969.131,E2 -17969.131} C_VEL
LIN {X 0,Y 270.267,Z 78.818,A -85,B 0,C 180,E1 -17972.146,E2 -17972.146} C_VEL
LIN {X 0,Y 270.28,Z 78.814,A -85,B 0,C 180,E1 -17975.519,E2 -17975.519} C_VEL
LIN {X 0,Y 270.305,Z 78.813,A -85,B 0,C 180,E1 -17980.245,E2 -17980.245} C_VEL
LIN {X 0,Y 270.407,Z 78.793,A -85,B 0,C 180,E1 -17984.936,E2 -17984.936} C_VEL
LIN {X 0,Y 270.414,Z 78.799,A -85,B 0,C 180,E1 -17989.518,E2 -17989.518} C_VEL
LIN {X 0,Y 270.432,Z 78.795,A -85,B 0,C 180,E1 -17989.887,E2 -17989.887} C_VEL
LIN {X 0,Y 270.151,Z 78.832,A -85,B 0,C 180,E1 -17990.719,E2 -17990.719} C_VEL
LIN {X 0,Y 268.803,Z 79,A -85,B 0,C 180,E1 -17991.947,E2 -17991.947} C_VEL
LIN {X 0,Y 264.467,Z 79.526,A -85,B 0,C 180,E1 -17994.806,E2 -17994.806} C_VEL
LIN {X 0,Y 263.517,Z 79.645,A -85,B 0,C 180,E1 -17996.085,E2 -17996.085} C_VEL
LIN {X 0,Y 263.492,Z 79.647,A -85,B 0,C 180,E1 -17996.518,E2 -17996.518} C_VEL
LIN {X 0,Y 263.754,Z 79.626,A -85,B 0,C 180,E1 -17998.473,E2 -17998.473} C_VEL
LIN {X 0,Y 263.754,Z 79.631,A -85,B 0,C 180,E1 -18001.527,E2 -18001.527} C_VEL
LIN {X 0,Y 263.534,Z 79.659,A -85,B 0,C 180,E1 -18007.663,E2 -18007.663} C_VEL
LIN {X 0,Y 263.353,Z 79.676,A -85,B 0,C 180,E1 -18010.767,E2 -18010.767} C_VEL
LIN {X 0,Y 263.327,Z 79.682,A -85,B 0,C 180,E1 -18015.48,E2 -18015.48} C_VEL
LIN {X 0,Y 263.266,Z 79.688,A -85,B 0,C 180,E1 -18020.307,E2 -18020.307} C_VEL
LIN {X 0,Y 263.181,Z 79.702,A -85,B 0,C 180,E1 -18025.294,E2 -18025.294} C_VEL
LIN {X 0,Y 263.142,Z 79.71,A -85,B 0,C 180,E1 -18028.734,E2 -18028.734} C_VEL
LIN {X 0,Y 263.131,Z 79.709,A -85,B 0,C 180,E1 -18032.289,E2 -18032.289} C_VEL
LIN {X 0,Y 263.186,Z 79.703,A -85,B 0,C 180,E1 -18036.763,E2 -18036.763} C_VEL
LIN {X 0,Y 263.127,Z 79.708,A -85,B 0,C 180,E1 -18041.593,E2 -18041.593} C_VEL
LIN {X 0,Y 263.125,Z 79.709,A -85,B 0,C 180,E1 -18046.016,E2 -18046.016} C_VEL
LIN {X 0,Y 263.108,Z 79.713,A -85,B 0,C 180,E1 -18050.127,E2 -18050.127} C_VEL
LIN {X 0,Y 263.172,Z 79.701,A -85,B 0,C 180,E1 -18054.019,E2 -18054.019} C_VEL
LIN {X 0,Y 263.216,Z 79.913,A -85,B 0,C 180,E1 -18054.956,E2 -18054.956} C_VEL
LIN {X 0,Y 265.361,Z 89.563,A -85,B 0,C 180,E1 -18058.26,E2 -18058.26} C_VEL
LIN {X 0,Y 267.643,Z 101.178,A -85,B 0,C 180,E1 -18062.035,E2 -18062.035} C_VEL
LIN {X 0,Y 267.632,Z 101.97,A -85,B 0,C 180,E1 -18062.255,E2 -18062.255} C_VEL
LIN {X 0,Y 271.414,Z 129.479,A -85,B 0,C 180,E1 -18063.377,E2 -18063.377} C_VEL
LIN {X 0,Y 274.032,Z 154.819,A -85,B 0,C 180,E1 -18064.306,E2 -18064.306} C_VEL
LIN {X 0,Y 272.559,Z 211.083,A -85,B 0,C 180,E1 -18065.786,E2 -18065.786} C_VEL
LIN {X 0,Y 271.691,Z 224.345,A -85,B 0,C 180,E1 -18066.413,E2 -18066.413} C_VEL
LIN {X 0,Y 270.48,Z 236.51,A -85,B 0,C 180,E1 -18067.263,E2 -18067.263} C_VEL
LIN {X 0,Y 269.087,Z 247.982,A -85,B 0,C 180,E1 -18068.351,E2 -18068.351} C_VEL
LIN {X 0,Y 267.452,Z 259.78,A -85,B 0,C 180,E1 -18069.824,E2 -18069.824} C_VEL
LIN {X 0,Y 266.103,Z 269.307,A -85,B 0,C 180,E1 -18071.323,E2 -18071.323} C_VEL
LIN {X 0,Y 264.45,Z 279.307,A -85,B 0,C 180,E1 -18073.261,E2 -18073.261} C_VEL
LIN {X 0,Y 263.839,Z 284.778,A -85,B 0,C 180,E1 -18074.551,E2 -18074.551} C_VEL
LIN {X 0,Y 262.683,Z 293.023,A -85,B 0,C 180,E1 -18076.855,E2 -18076.855} C_VEL
LIN {X 0,Y 261.854,Z 299.646,A -85,B 0,C 180,E1 -18079.171,E2 -18079.171} C_VEL
LIN {X 0,Y 261.418,Z 304.909,A -85,B 0,C 180,E1 -18081.497,E2 -18081.497} C_VEL
LIN {X 0,Y 261.223,Z 308.979,A -85,B 0,C 180,E1 -18083.822,E2 -18083.822} C_VEL
LIN {X 0,Y 261.234,Z 311.075,A -85,B 0,C 180,E1 -18085.371,E2 -18085.371} C_VEL
LIN {X 0,Y 261.308,Z 312.735,A -85,B 0,C 180,E1 -18086.916,E2 -18086.916} C_VEL
LIN {X 0,Y 261.322,Z 313.976,A -85,B 0,C 180,E1 -18088.459,E2 -18088.459} C_VEL
LIN {X 0,Y 261.392,Z 314.8,A -85,B 0,C 180,E1 -18090,E2 -18090} C_VEL
LIN {X 0,Y 261.241,Z 315.16,A -85,B 0,C 180,E1 -18093.084,E2 -18093.084} C_VEL
LIN {X 0,Y 261.144,Z 313.962,A -85,B 0,C 180,E1 -18096.18,E2 -18096.18} C_VEL
LIN {X 0,Y 261.581,Z 311.102,A -85,B 0,C 180,E1 -18099.277,E2 -18099.277} C_VEL
LIN {X 0,Y 262.223,Z 307.858,A -85,B 0,C 180,E1 -18101.596,E2 -18101.596} C_VEL
LIN {X 0,Y 263.363,Z 303.575,A -85,B 0,C 180,E1 -18103.897,E2 -18103.897} C_VEL
LIN {X 0,Y 264.978,Z 298.136,A -85,B 0,C 180,E1 -18106.17,E2 -18106.17} C_VEL
LIN {X 0,Y 266.9,Z 291.362,A -85,B 0,C 180,E1 -18108.42,E2 -18108.42} C_VEL
LIN {X 0,Y 269.189,Z 282.992,A -85,B 0,C 180,E1 -18110.638,E2 -18110.638} C_VEL
LIN {X 0,Y 271.587,Z 274.403,A -85,B 0,C 180,E1 -18112.439,E2 -18112.439} C_VEL
LIN {X 0,Y 274.322,Z 263.848,A -85,B 0,C 180,E1 -18114.199,E2 -18114.199} C_VEL
LIN {X 0,Y 276.684,Z 253.411,A -85,B 0,C 180,E1 -18115.583,E2 -18115.583} C_VEL
LIN {X 0,Y 278.951,Z 241.938,A -85,B 0,C 180,E1 -18116.766,E2 -18116.766} C_VEL
LIN {X 0,Y 280.826,Z 230.073,A -85,B 0,C 180,E1 -18117.681,E2 -18117.681} C_VEL
LIN {X 0,Y 282.388,Z 216.197,A -85,B 0,C 180,E1 -18118.435,E2 -18118.435} C_VEL
LIN {X 0,Y 283.306,Z 203.145,A -85,B 0,C 180,E1 -18118.855,E2 -18118.855} C_VEL
LIN {X 0,Y 284.795,Z 156.598,A -85,B 0,C 180,E1 -18120.043,E2 -18120.043} C_VEL
LIN {X 0,Y 281.252,Z 133.742,A -85,B 0,C 180,E1 -18121.222,E2 -18121.222} C_VEL
LIN {X 0,Y 278.742,Z 121.75,A -85,B 0,C 180,E1 -18121.955,E2 -18121.955} C_VEL
LIN {X 0,Y 270.554,Z 104.496,A -85,B 0,C 180,E1 -18123.773,E2 -18123.773} C_VEL
LIN {X 0,Y 268.522,Z 100.179,A -85,B 0,C 180,E1 -18124.302,E2 -18124.302} C_VEL
LIN {X 0,Y 266.456,Z 91.535,A -85,B 0,C 180,E1 -18127.695,E2 -18127.695} C_VEL
LIN {X 0,Y 264.093,Z 83.201,A -85,B 0,C 180,E1 -18131.254,E2 -18131.254} C_VEL
LIN {X 0,Y 263.131,Z 79.703,A -85,B 0,C 180,E1 -18132.874,E2 -18132.874} C_VEL
LIN {X 0,Y 263.126,Z 79.704,A -85,B 0,C 180,E1 -18136.151,E2 -18136.151} C_VEL
LIN {X 0,Y 263.108,Z 79.699,A -85,B 0,C 180,E1 -18140.128,E2 -18140.128} C_VEL
LIN {X 0,Y 263.166,Z 79.697,A -85,B 0,C 180,E1 -18144.018,E2 -18144.018} C_VEL
LIN {X 0,Y 263.135,Z 79.705,A -85,B 0,C 180,E1 -18147.712,E2 -18147.712} C_VEL
LIN {X 0,Y 263.204,Z 79.699,A -85,B 0,C 180,E1 -18151.783,E2 -18151.783} C_VEL
LIN {X 0,Y 263.229,Z 79.692,A -85,B 0,C 180,E1 -18155.2,E2 -18155.2} C_VEL
LIN {X 0,Y 263.266,Z 79.688,A -85,B 0,C 180,E1 -18159.693,E2 -18159.693} C_VEL
LIN {X 0,Y 263.354,Z 79.676,A -85,B 0,C 180,E1 -18164.522,E2 -18164.522} C_VEL
LIN {X 0,Y 263.358,Z 79.675,A -85,B 0,C 180,E1 -18169.234,E2 -18169.234} C_VEL
LIN {X 0,Y 263.561,Z 79.642,A -85,B 0,C 180,E1 -18172.338,E2 -18172.338} C_VEL
LIN {X 0,Y 263.753,Z 79.617,A -85,B 0,C 180,E1 -18178.473,E2 -18178.473} C_VEL
LIN {X 0,Y 263.753,Z 79.631,A -85,B 0,C 180,E1 -18181.527,E2 -18181.527} C_VEL
LIN {X 0,Y 263.546,Z 79.649,A -85,B 0,C 180,E1 -18187.662,E2 -18187.662} C_VEL
LIN {X 0,Y 263.355,Z 79.678,A -85,B 0,C 180,E1 -18190.766,E2 -18190.766} C_VEL
LIN {X 0,Y 263.326,Z 79.681,A -85,B 0,C 180,E1 -18195.479,E2 -18195.479} C_VEL
LIN {X 0,Y 263.264,Z 79.69,A -85,B 0,C 180,E1 -18200.306,E2 -18200.306} C_VEL
LIN {X 0,Y 263.179,Z 79.703,A -85,B 0,C 180,E1 -18205.294,E2 -18205.294} C_VEL
LIN {X 0,Y 263.14,Z 79.708,A -85,B 0,C 180,E1 -18208.734,E2 -18208.734} C_VEL
LIN {X 0,Y 263.129,Z 79.709,A -85,B 0,C 180,E1 -18212.289,E2 -18212.289} C_VEL
LIN {X 0,Y 263.177,Z 79.698,A -85,B 0,C 180,E1 -18216.761,E2 -18216.761} C_VEL
LIN {X 0,Y 263.106,Z 79.697,A -85,B 0,C 180,E1 -18219.872,E2 -18219.872} C_VEL
LIN {X 0,Y 263.104,Z 79.712,A -85,B 0,C 180,E1 -18223.988,E2 -18223.988} C_VEL
LIN {X 0,Y 263.114,Z 79.712,A -85,B 0,C 180,E1 -18224.89,E2 -18224.89} C_VEL
LIN {X 0,Y 264.115,Z 82.578,A -85,B 0,C 180,E1 -18225.179,E2 -18225.179} C_VEL
LIN {X 0,Y 266.018,Z 85.184,A -85,B 0,C 180,E1 -18225.603,E2 -18225.603} C_VEL
LIN {X 0,Y 275.033,Z 99.737,A -85,B 0,C 180,E1 -18227.572,E2 -18227.572} C_VEL
LIN {X 0,Y 280.972,Z 111.149,A -85,B 0,C 180,E1 -18228.828,E2 -18228.828} C_VEL
LIN {X 0,Y 286.197,Z 122.488,A -85,B 0,C 180,E1 -18229.913,E2 -18229.913} C_VEL
LIN {X 0,Y 283.676,Z 184.657,A -85,B 0,C 180,E1 -18231.479,E2 -18231.479} C_VEL
LIN {X 0,Y 282.725,Z 197.57,A -85,B 0,C 180,E1 -18232.088,E2 -18232.088} C_VEL
LIN {X 0,Y 281.434,Z 210.18,A -85,B 0,C 180,E1 -18232.977,E2 -18232.977} C_VEL
LIN {X 0,Y 279.657,Z 221.63,A -85,B 0,C 180,E1 -18234.05,E2 -18234.05} C_VEL
LIN {X 0,Y 277.404,Z 233.252,A -85,B 0,C 180,E1 -18235.468,E2 -18235.468} C_VEL
LIN {X 0,Y 275.126,Z 243.822,A -85,B 0,C 180,E1 -18237.124,E2 -18237.124} C_VEL
LIN {X 0,Y 272.634,Z 253.216,A -85,B 0,C 180,E1 -18238.965,E2 -18238.965} C_VEL
LIN {X 0,Y 270.102,Z 262.282,A -85,B 0,C 180,E1 -18241.225,E2 -18241.225} C_VEL
LIN {X 0,Y 267.891,Z 269.515,A -85,B 0,C 180,E1 -18243.513,E2 -18243.513} C_VEL
LIN {X 0,Y 265.994,Z 275.217,A -85,B 0,C 180,E1 -18245.824,E2 -18245.824} C_VEL
LIN {X 0,Y 264.314,Z 280.253,A -85,B 0,C 180,E1 -18248.534,E2 -18248.534} C_VEL
LIN {X 0,Y 262.975,Z 283.88,A -85,B 0,C 180,E1 -18251.295,E2 -18251.295} C_VEL
LIN {X 0,Y 262.404,Z 285.292,A -85,B 0,C 180,E1 -18252.866,E2 -18252.866} C_VEL
LIN {X 0,Y 261.862,Z 286.577,A -85,B 0,C 180,E1 -18255.058,E2 -18255.058} C_VEL
LIN {X 0,Y 261.407,Z 287.06,A -85,B 0,C 180,E1 -18257.58,E2 -18257.58} C_VEL
LIN {X 0,Y 261.224,Z 286.176,A -85,B 0,C 180,E1 -18260.71,E2 -18260.71} C_VEL
LIN {X 0,Y 261.589,Z 283.787,A -85,B 0,C 180,E1 -18263.753,E2 -18263.753} C_VEL
LIN {X 0,Y 261.755,Z 280.746,A -85,B 0,C 180,E1 -18266.151,E2 -18266.151} C_VEL
LIN {X 0,Y 262.273,Z 276.743,A -85,B 0,C 180,E1 -18268.465,E2 -18268.465} C_VEL
LIN {X 0,Y 263.036,Z 270.604,A -85,B 0,C 180,E1 -18271.148,E2 -18271.148} C_VEL
LIN {X 0,Y 264.132,Z 263.905,A -85,B 0,C 180,E1 -18273.432,E2 -18273.432} C_VEL
LIN {X 0,Y 265.403,Z 255.613,A -85,B 0,C 180,E1 -18275.699,E2 -18275.699} C_VEL
LIN {X 0,Y 266.656,Z 247.08,A -85,B 0,C 180,E1 -18277.573,E2 -18277.573} C_VEL
LIN {X 0,Y 268.267,Z 237.677,A -85,B 0,C 180,E1 -18279.234,E2 -18279.234} C_VEL
LIN {X 0,Y 269.841,Z 226.056,A -85,B 0,C 180,E1 -18280.885,E2 -18280.885} C_VEL
LIN {X 0,Y 271.113,Z 214.52,A -85,B 0,C 180,E1 -18282.159,E2 -18282.159} C_VEL
LIN {X 0,Y 272.088,Z 202.583,A -85,B 0,C 180,E1 -18283.158,E2 -18283.158} C_VEL
LIN {X 0,Y 272.861,Z 189.643,A -85,B 0,C 180,E1 -18283.926,E2 -18283.926} C_VEL
LIN {X 0,Y 273.328,Z 177.407,A -85,B 0,C 180,E1 -18284.376,E2 -18284.376} C_VEL
LIN {X 0,Y 275.035,Z 109.23,A -85,B 0,C 180,E1 -18286.128,E2 -18286.128} C_VEL
LIN {X 0,Y 269.755,Z 94.512,A -85,B 0,C 180,E1 -18287.015,E2 -18287.015} C_VEL
LIN {X 0,Y 263.422,Z 80.453,A -85,B 0,C 180,E1 -18288.026,E2 -18288.026} C_VEL
LIN {X 0,Y 263.266,Z 79.692,A -85,B 0,C 180,E1 -18288.072,E2 -18288.072} C_VEL
LIN {X 0,Y 263.215,Z 79.692,A -85,B 0,C 180,E1 -18290.849,E2 -18290.849} C_VEL
LIN {X 0,Y 263.194,Z 79.699,A -85,B 0,C 180,E1 -18295.293,E2 -18295.293} C_VEL
LIN {X 0,Y 263.167,Z 79.703,A -85,B 0,C 180,E1 -18298.731,E2 -18298.731} C_VEL
LIN {X 0,Y 263.135,Z 79.709,A -85,B 0,C 180,E1 -18302.288,E2 -18302.288} C_VEL
LIN {X 0,Y 263.192,Z 79.702,A -85,B 0,C 180,E1 -18305.978,E2 -18305.978} C_VEL
LIN {X 0,Y 263.123,Z 79.709,A -85,B 0,C 180,E1 -18309.87,E2 -18309.87} C_VEL
LIN {X 0,Y 263.125,Z 79.707,A -85,B 0,C 180,E1 -18313.984,E2 -18313.984} C_VEL
LIN {X 0,Y 263.126,Z 79.705,A -85,B 0,C 180,E1 -18318.407,E2 -18318.407} C_VEL
LIN {X 0,Y 263.185,Z 79.7,A -85,B 0,C 180,E1 -18323.237,E2 -18323.237} C_VEL
LIN {X 0,Y 263.135,Z 79.705,A -85,B 0,C 180,E1 -18327.712,E2 -18327.712} C_VEL
LIN {X 0,Y 263.203,Z 79.697,A -85,B 0,C 180,E1 -18331.784,E2 -18331.784} C_VEL
LIN {X 0,Y 263.229,Z 79.693,A -85,B 0,C 180,E1 -18335.201,E2 -18335.201} C_VEL
LIN {X 0,Y 263.267,Z 79.688,A -85,B 0,C 180,E1 -18339.694,E2 -18339.694} C_VEL
LIN {X 0,Y 263.354,Z 79.666,A -85,B 0,C 180,E1 -18344.522,E2 -18344.522} C_VEL
LIN {X 0,Y 263.357,Z 79.678,A -85,B 0,C 180,E1 -18349.234,E2 -18349.234} C_VEL
LIN {X 0,Y 263.559,Z 79.649,A -85,B 0,C 180,E1 -18352.338,E2 -18352.338} C_VEL
LIN {X 0,Y 263.492,Z 79.647,A -85,B 0,C 180,E1 -18356.518,E2 -18356.518} C_VEL
LIN {X 0,Y 262.989,Z 79.719,A -85,B 0,C 180,E1 -18357.796,E2 -18357.796} C_VEL
LIN {X 0,Y 261.508,Z 79.911,A -85,B 0,C 180,E1 -18359.052,E2 -18359.052} C_VEL
LIN {X 0,Y 256.893,Z 80.487,A -85,B 0,C 180,E1 -18362.446,E2 -18362.446} C_VEL
LIN {X 0,Y 256.467,Z 80.535,A -85,B 0,C 180,E1 -18363.335,E2 -18363.335} C_VEL
LIN {X 0,Y 256.497,Z 80.534,A -85,B 0,C 180,E1 -18367.874,E2 -18367.874} C_VEL
LIN {X 0,Y 256.294,Z 80.556,A -85,B 0,C 180,E1 -18371.067,E2 -18371.067} C_VEL
LIN {X 0,Y 256.263,Z 80.561,A -85,B 0,C 180,E1 -18375.918,E2 -18375.918} C_VEL
LIN {X 0,Y 256.168,Z 80.574,A -85,B 0,C 180,E1 -18380.895,E2 -18380.895} C_VEL
LIN {X 0,Y 256.166,Z 80.576,A -85,B 0,C 180,E1 -18385.126,E2 -18385.126} C_VEL
LIN {X 0,Y 256.06,Z 80.589,A -85,B 0,C 180,E1 -18389.607,E2 -18389.607} C_VEL
LIN {X 0,Y 256.069,Z 80.588,A -85,B 0,C 180,E1 -18393.293,E2 -18393.293} C_VEL
LIN {X 0,Y 256.118,Z 80.581,A -85,B 0,C 180,E1 -18397.271,E2 -18397.271} C_VEL
LIN {X 0,Y 256.057,Z 80.588,A -85,B 0,C 180,E1 -18401.203,E2 -18401.203} C_VEL
LIN {X 0,Y 256.06,Z 80.588,A -85,B 0,C 180,E1 -18405.53,E2 -18405.53} C_VEL
LIN {X 0,Y 256.057,Z 80.591,A -85,B 0,C 180,E1 -18408.796,E2 -18408.796} C_VEL
LIN {X 0,Y 256.132,Z 80.58,A -85,B 0,C 180,E1 -18412.867,E2 -18412.867} C_VEL
LIN {X 0,Y 256.152,Z 80.673,A -85,B 0,C 180,E1 -18414.396,E2 -18414.396} C_VEL
LIN {X 0,Y 258.154,Z 89.593,A -85,B 0,C 180,E1 -18417.56,E2 -18417.56} C_VEL
LIN {X 0,Y 260.568,Z 101.555,A -85,B 0,C 180,E1 -18421.569,E2 -18421.569} C_VEL
LIN {X 0,Y 261.747,Z 106.951,A -85,B 0,C 180,E1 -18421.844,E2 -18421.844} C_VEL
LIN {X 0,Y 265.642,Z 137.482,A -85,B 0,C 180,E1 -18423.096,E2 -18423.096} C_VEL
LIN {X 0,Y 267.451,Z 155.163,A -85,B 0,C 180,E1 -18423.762,E2 -18423.762} C_VEL
LIN {X 0,Y 265.957,Z 210.504,A -85,B 0,C 180,E1 -18425.249,E2 -18425.249} C_VEL
LIN {X 0,Y 265.059,Z 223.831,A -85,B 0,C 180,E1 -18425.889,E2 -18425.889} C_VEL
LIN {X 0,Y 263.803,Z 236.029,A -85,B 0,C 180,E1 -18426.757,E2 -18426.757} C_VEL
LIN {X 0,Y 262.247,Z 248.337,A -85,B 0,C 180,E1 -18427.964,E2 -18427.964} C_VEL
LIN {X 0,Y 260.555,Z 259.991,A -85,B 0,C 180,E1 -18429.473,E2 -18429.473} C_VEL
LIN {X 0,Y 259.028,Z 270.504,A -85,B 0,C 180,E1 -18431.204,E2 -18431.204} C_VEL
LIN {X 0,Y 257.442,Z 279.391,A -85,B 0,C 180,E1 -18433.013,E2 -18433.013} C_VEL
LIN {X 0,Y 256.687,Z 285.488,A -85,B 0,C 180,E1 -18434.517,E2 -18434.517} C_VEL
LIN {X 0,Y 255.528,Z 293.542,A -85,B 0,C 180,E1 -18436.885,E2 -18436.885} C_VEL
LIN {X 0,Y 254.83,Z 298.982,A -85,B 0,C 180,E1 -18438.869,E2 -18438.869} C_VEL
LIN {X 0,Y 254.348,Z 304.305,A -85,B 0,C 180,E1 -18441.259,E2 -18441.259} C_VEL
LIN {X 0,Y 254.147,Z 308.428,A -85,B 0,C 180,E1 -18443.649,E2 -18443.649} C_VEL
LIN {X 0,Y 254.144,Z 310.568,A -85,B 0,C 180,E1 -18445.241,E2 -18445.241} C_VEL
LIN {X 0,Y 254.234,Z 312.252,A -85,B 0,C 180,E1 -18446.83,E2 -18446.83} C_VEL
LIN {X 0,Y 254.243,Z 313.515,A -85,B 0,C 180,E1 -18448.416,E2 -18448.416} C_VEL
LIN {X 0,Y 254.306,Z 314.374,A -85,B 0,C 180,E1 -18450,E2 -18450} C_VEL
LIN {X 0,Y 254.185,Z 314.778,A -85,B 0,C 180,E1 -18451.584,E2 -18451.584} C_VEL
LIN {X 0,Y 254.144,Z 314.785,A -85,B 0,C 180,E1 -18453.17,E2 -18453.17} C_VEL
LIN {X 0,Y 254.087,Z 314.21,A -85,B 0,C 180,E1 -18455.279,E2 -18455.279} C_VEL
LIN {X 0,Y 254.232,Z 312.445,A -85,B 0,C 180,E1 -18457.945,E2 -18457.945} C_VEL
LIN {X 0,Y 254.725,Z 309.904,A -85,B 0,C 180,E1 -18460.331,E2 -18460.331} C_VEL
LIN {X 0,Y 255.534,Z 306.369,A -85,B 0,C 180,E1 -18462.711,E2 -18462.711} C_VEL
LIN {X 0,Y 257.001,Z 301.772,A -85,B 0,C 180,E1 -18465.058,E2 -18465.058} C_VEL
LIN {X 0,Y 259.118,Z 294.89,A -85,B 0,C 180,E1 -18467.751,E2 -18467.751} C_VEL
LIN {X 0,Y 261.259,Z 287.389,A -85,B 0,C 180,E1 -18470.058,E2 -18470.058} C_VEL
LIN {X 0,Y 263.486,Z 279.809,A -85,B 0,C 180,E1 -18471.927,E2 -18471.927} C_VEL
LIN {X 0,Y 266.117,Z 270.661,A -85,B 0,C 180,E1 -18473.75,E2 -18473.75} C_VEL
LIN {X 0,Y 268.692,Z 260.532,A -85,B 0,C 180,E1 -18475.36,E2 -18475.36} C_VEL
LIN {X 0,Y 271.298,Z 249.314,A -85,B 0,C 180,E1 -18476.75,E2 -18476.75} C_VEL
LIN {X 0,Y 273.685,Z 236.729,A -85,B 0,C 180,E1 -18477.946,E2 -18477.946} C_VEL
LIN {X 0,Y 275.592,Z 223.728,A -85,B 0,C 180,E1 -18478.825,E2 -18478.825} C_VEL
LIN {X 0,Y 276.841,Z 210.974,A -85,B 0,C 180,E1 -18479.41,E2 -18479.41} C_VEL
LIN {X 0,Y 278.064,Z 183.725,A -85,B 0,C 180,E1 -18480.137,E2 -18480.137} C_VEL
LIN {X 0,Y 278.912,Z 157.82,A -85,B 0,C 180,E1 -18480.814,E2 -18480.814} C_VEL
LIN {X 0,Y 275.391,Z 134.98,A -85,B 0,C 180,E1 -18482.036,E2 -18482.036} C_VEL
LIN {X 0,Y 273.353,Z 125.002,A -85,B 0,C 180,E1 -18482.663,E2 -18482.663} C_VEL
LIN {X 0,Y 265.584,Z 108.438,A -85,B 0,C 180,E1 -18484.467,E2 -18484.467} C_VEL
LIN {X 0,Y 261.241,Z 99.732,A -85,B 0,C 180,E1 -18485.56,E2 -18485.56} C_VEL
LIN {X 0,Y 259.238,Z 91.506,A -85,B 0,C 180,E1 -18488.948,E2 -18488.948} C_VEL
LIN {X 0,Y 256.454,Z 82.084,A -85,B 0,C 180,E1 -18493.245,E2 -18493.245} C_VEL
LIN {X 0,Y 256.081,Z 80.581,A -85,B 0,C 180,E1 -18493.984,E2 -18493.984} C_VEL
LIN {X 0,Y 256.074,Z 80.578,A -85,B 0,C 180,E1 -18497.819,E2 -18497.819} C_VEL
LIN {X 0,Y 256.073,Z 80.578,A -85,B 0,C 180,E1 -18500.858,E2 -18500.858} C_VEL
LIN {X 0,Y 256.133,Z 80.569,A -85,B 0,C 180,E1 -18502.868,E2 -18502.868} C_VEL
LIN {X 0,Y 256.07,Z 80.578,A -85,B 0,C 180,E1 -18506.707,E2 -18506.707} C_VEL
LIN {X 0,Y 256.116,Z 80.573,A -85,B 0,C 180,E1 -18510.4,E2 -18510.4} C_VEL
LIN {X 0,Y 256.191,Z 80.565,A -85,B 0,C 180,E1 -18514.861,E2 -18514.861} C_VEL
LIN {X 0,Y 256.169,Z 80.567,A -85,B 0,C 180,E1 -18519.105,E2 -18519.105} C_VEL
LIN {X 0,Y 256.303,Z 80.551,A -85,B 0,C 180,E1 -18524.085,E2 -18524.085} C_VEL
LIN {X 0,Y 256.298,Z 80.547,A -85,B 0,C 180,E1 -18527.328,E2 -18527.328} C_VEL
LIN {X 0,Y 256.518,Z 80.521,A -85,B 0,C 180,E1 -18532.126,E2 -18532.126} C_VEL
LIN {X 0,Y 256.499,Z 80.531,A -85,B 0,C 180,E1 -18536.858,E2 -18536.858} C_VEL
LIN {X 0,Y 256.768,Z 80.496,A -85,B 0,C 180,E1 -18540,E2 -18540} C_VEL
LIN {X 0,Y 256.498,Z 80.522,A -85,B 0,C 180,E1 -18543.141,E2 -18543.141} C_VEL
LIN {X 0,Y 256.506,Z 80.524,A -85,B 0,C 180,E1 -18547.874,E2 -18547.874} C_VEL
LIN {X 0,Y 256.29,Z 80.555,A -85,B 0,C 180,E1 -18552.672,E2 -18552.672} C_VEL
LIN {X 0,Y 256.245,Z 80.566,A -85,B 0,C 180,E1 -18556.271,E2 -18556.271} C_VEL
LIN {X 0,Y 256.167,Z 80.578,A -85,B 0,C 180,E1 -18560.895,E2 -18560.895} C_VEL
LIN {X 0,Y 256.164,Z 80.577,A -85,B 0,C 180,E1 -18565.126,E2 -18565.126} C_VEL
LIN {X 0,Y 256.059,Z 80.589,A -85,B 0,C 180,E1 -18569.606,E2 -18569.606} C_VEL
LIN {X 0,Y 256.067,Z 80.585,A -85,B 0,C 180,E1 -18573.293,E2 -18573.293} C_VEL
LIN {X 0,Y 256.111,Z 80.578,A -85,B 0,C 180,E1 -18577.269,E2 -18577.269} C_VEL
LIN {X 0,Y 256.054,Z 80.57,A -85,B 0,C 180,E1 -18581.203,E2 -18581.203} C_VEL
LIN {X 0,Y 256.061,Z 80.617,A -85,B 0,C 180,E1 -18583.611,E2 -18583.611} C_VEL
LIN {X 0,Y 256.99,Z 83.276,A -85,B 0,C 180,E1 -18583.887,E2 -18583.887} C_VEL
LIN {X 0,Y 258.952,Z 85.878,A -85,B 0,C 180,E1 -18584.353,E2 -18584.353} C_VEL
LIN {X 0,Y 268.541,Z 101.226,A -85,B 0,C 180,E1 -18586.573,E2 -18586.573} C_VEL
LIN {X 0,Y 273.713,Z 110.595,A -85,B 0,C 180,E1 -18587.715,E2 -18587.715} C_VEL
LIN {X 0,Y 280.263,Z 124.539,A -85,B 0,C 180,E1 -18589.139,E2 -18589.139} C_VEL
LIN {X 0,Y 277.723,Z 185.312,A -85,B 0,C 180,E1 -18590.706,E2 -18590.706} C_VEL
LIN {X 0,Y 276.688,Z 198.441,A -85,B 0,C 180,E1 -18591.34,E2 -18591.34} C_VEL
LIN {X 0,Y 275.375,Z 210.695,A -85,B 0,C 180,E1 -18592.228,E2 -18592.228} C_VEL
LIN {X 0,Y 273.43,Z 222.584,A -85,B 0,C 180,E1 -18593.372,E2 -18593.372} C_VEL
LIN {X 0,Y 271.146,Z 233.846,A -85,B 0,C 180,E1 -18594.78,E2 -18594.78} C_VEL
LIN {X 0,Y 268.769,Z 244.376,A -85,B 0,C 180,E1 -18596.468,E2 -18596.468} C_VEL
LIN {X 0,Y 266.416,Z 252.904,A -85,B 0,C 180,E1 -18598.157,E2 -18598.157} C_VEL
LIN {X 0,Y 263.717,Z 262.09,A -85,B 0,C 180,E1 -18600.461,E2 -18600.461} C_VEL
LIN {X 0,Y 261.368,Z 269.439,A -85,B 0,C 180,E1 -18602.799,E2 -18602.799} C_VEL
LIN {X 0,Y 259.352,Z 275.258,A -85,B 0,C 180,E1 -18605.164,E2 -18605.164} C_VEL
LIN {X 0,Y 257.734,Z 279.785,A -85,B 0,C 180,E1 -18607.557,E2 -18607.557} C_VEL
LIN {X 0,Y 256.89,Z 282.151,A -85,B 0,C 180,E1 -18609.166,E2 -18609.166} C_VEL
LIN {X 0,Y 256.093,Z 284.076,A -85,B 0,C 180,E1 -18610.773,E2 -18610.773} C_VEL
LIN {X 0,Y 255.471,Z 285.56,A -85,B 0,C 180,E1 -18612.386,E2 -18612.386} C_VEL
LIN {X 0,Y 254.827,Z 286.982,A -85,B 0,C 180,E1 -18614.858,E2 -18614.858} C_VEL
LIN {X 0,Y 254.372,Z 287.438,A -85,B 0,C 180,E1 -18617.23,E2 -18617.23} C_VEL
LIN {X 0,Y 254.168,Z 287.257,A -85,B 0,C 180,E1 -18618.84,E2 -18618.84} C_VEL
LIN {X 0,Y 254.22,Z 285.656,A -85,B 0,C 180,E1 -18622.055,E2 -18622.055} C_VEL
LIN {X 0,Y 254.498,Z 284.122,A -85,B 0,C 180,E1 -18623.797,E2 -18623.797} C_VEL
LIN {X 0,Y 254.67,Z 281.365,A -85,B 0,C 180,E1 -18626.044,E2 -18626.044} C_VEL
LIN {X 0,Y 255.184,Z 277.437,A -85,B 0,C 180,E1 -18628.422,E2 -18628.422} C_VEL
LIN {X 0,Y 255.789,Z 272.4,A -85,B 0,C 180,E1 -18630.787,E2 -18630.787} C_VEL
LIN {X 0,Y 256.838,Z 266.044,A -85,B 0,C 180,E1 -18633.137,E2 -18633.137} C_VEL
LIN {X 0,Y 258.114,Z 258.118,A -85,B 0,C 180,E1 -18635.469,E2 -18635.469} C_VEL
LIN {X 0,Y 259.665,Z 248.276,A -85,B 0,C 180,E1 -18637.778,E2 -18637.778} C_VEL
LIN {X 0,Y 261.319,Z 239.057,A -85,B 0,C 180,E1 -18639.482,E2 -18639.482} C_VEL
LIN {X 0,Y 262.729,Z 229.07,A -85,B 0,C 180,E1 -18640.988,E2 -18640.988} C_VEL
LIN {X 0,Y 264.07,Z 218.211,A -85,B 0,C 180,E1 -18642.293,E2 -18642.293} C_VEL
LIN {X 0,Y 265.157,Z 206.265,A -85,B 0,C 180,E1 -18643.41,E2 -18643.41} C_VEL
LIN {X 0,Y 266.01,Z 194.006,A -85,B 0,C 180,E1 -18644.243,E2 -18644.243} C_VEL
LIN {X 0,Y 266.598,Z 181.374,A -85,B 0,C 180,E1 -18644.796,E2 -18644.796} C_VEL
LIN {X 0,Y 268.487,Z 110.681,A -85,B 0,C 180,E1 -18646.669,E2 -18646.669} C_VEL
LIN {X 0,Y 263.66,Z 97.395,A -85,B 0,C 180,E1 -18647.505,E2 -18647.505} C_VEL
LIN {X 0,Y 256.332,Z 81.166,A -85,B 0,C 180,E1 -18648.724,E2 -18648.724} C_VEL
LIN {X 0,Y 256.216,Z 80.57,A -85,B 0,C 180,E1 -18648.788,E2 -18648.788} C_VEL
LIN {X 0,Y 256.085,Z 80.586,A -85,B 0,C 180,E1 -18652.595,E2 -18652.595} C_VEL
LIN {X 0,Y 256.131,Z 80.582,A -85,B 0,C 180,E1 -18656.042,E2 -18656.042} C_VEL
LIN {X 0,Y 256.105,Z 80.584,A -85,B 0,C 180,E1 -18659.601,E2 -18659.601} C_VEL
LIN {X 0,Y 256.086,Z 80.585,A -85,B 0,C 180,E1 -18663.29,E2 -18663.29} C_VEL
LIN {X 0,Y 256.13,Z 80.579,A -85,B 0,C 180,E1 -18667.275,E2 -18667.275} C_VEL
LIN {X 0,Y 256.064,Z 80.587,A -85,B 0,C 180,E1 -18671.202,E2 -18671.202} C_VEL
LIN {X 0,Y 256.046,Z 80.588,A -85,B 0,C 180,E1 -18675.534,E2 -18675.534} C_VEL
LIN {X 0,Y 256.056,Z 80.587,A -85,B 0,C 180,E1 -18678.797,E2 -18678.797} C_VEL
LIN {X 0,Y 256.133,Z 80.579,A -85,B 0,C 180,E1 -18682.868,E2 -18682.868} C_VEL
LIN {X 0,Y 256.07,Z 80.587,A -85,B 0,C 180,E1 -18686.708,E2 -18686.708} C_VEL
LIN {X 0,Y 256.116,Z 80.578,A -85,B 0,C 180,E1 -18690.401,E2 -18690.401} C_VEL
LIN {X 0,Y 256.191,Z 80.57,A -85,B 0,C 180,E1 -18694.862,E2 -18694.862} C_VEL
LIN {X 0,Y 256.171,Z 80.573,A -85,B 0,C 180,E1 -18699.105,E2 -18699.105} C_VEL
LIN {X 0,Y 256.303,Z 80.54,A -85,B 0,C 180,E1 -18704.085,E2 -18704.085} C_VEL
LIN {X 0,Y 256.299,Z 80.558,A -85,B 0,C 180,E1 -18708.934,E2 -18708.934} C_VEL
LIN {X 0,Y 256.517,Z 80.528,A -85,B 0,C 180,E1 -18712.127,E2 -18712.127} C_VEL
LIN {X 0,Y 256.498,Z 80.522,A -85,B 0,C 180,E1 -18716.859,E2 -18716.859} C_VEL
LIN {X 0,Y 256.769,Z 80.501,A -85,B 0,C 180,E1 -18720,E2 -18720} C_VEL
LIN {X 0,Y 256.467,Z 80.535,A -85,B 0,C 180,E1 -18723.335,E2 -18723.335} C_VEL
LIN {X 0,Y 255.679,Z 80.631,A -85,B 0,C 180,E1 -18724.645,E2 -18724.645} C_VEL
LIN {X 0,Y 252.827,Z 80.99,A -85,B 0,C 180,E1 -18726.784,E2 -18726.784} C_VEL
LIN {X 0,Y 249.641,Z 81.387,A -85,B 0,C 180,E1 -18729.418,E2 -18729.418} C_VEL
LIN {X 0,Y 249.283,Z 81.427,A -85,B 0,C 180,E1 -18730.328,E2 -18730.328} C_VEL
LIN {X 0,Y 249.186,Z 81.443,A -85,B 0,C 180,E1 -18734.705,E2 -18734.705} C_VEL
LIN {X 0,Y 249.125,Z 81.452,A -85,B 0,C 180,E1 -18738.079,E2 -18738.079} C_VEL
LIN {X 0,Y 249.088,Z 81.458,A -85,B 0,C 180,E1 -18741.518,E2 -18741.518} C_VEL
LIN {X 0,Y 249.11,Z 81.454,A -85,B 0,C 180,E1 -18745.471,E2 -18745.471} C_VEL
LIN {X 0,Y 249.044,Z 81.466,A -85,B 0,C 180,E1 -18748.976,E2 -18748.976} C_VEL
LIN {X 0,Y 249.03,Z 81.467,A -85,B 0,C 180,E1 -18752.426,E2 -18752.426} C_VEL
LIN {X 0,Y 249.051,Z 81.464,A -85,B 0,C 180,E1 -18756.342,E2 -18756.342} C_VEL
LIN {X 0,Y 249.009,Z 81.469,A -85,B 0,C 180,E1 -18760.478,E2 -18760.478} C_VEL
LIN {X 0,Y 249.005,Z 81.467,A -85,B 0,C 180,E1 -18764.879,E2 -18764.879} C_VEL
LIN {X 0,Y 249.019,Z 81.467,A -85,B 0,C 180,E1 -18767.363,E2 -18767.363} C_VEL
LIN {X 0,Y 249.045,Z 81.464,A -85,B 0,C 180,E1 -18772.2,E2 -18772.2} C_VEL
LIN {X 0,Y 249.117,Z 81.545,A -85,B 0,C 180,E1 -18773.843,E2 -18773.843} C_VEL
LIN {X 0,Y 251.269,Z 91.235,A -85,B 0,C 180,E1 -18777.392,E2 -18777.392} C_VEL
LIN {X 0,Y 253.282,Z 101.025,A -85,B 0,C 180,E1 -18780.797,E2 -18780.797} C_VEL
LIN {X 0,Y 255.167,Z 107.23,A -85,B 0,C 180,E1 -18781.2,E2 -18781.2} C_VEL
LIN {X 0,Y 259.045,Z 137.638,A -85,B 0,C 180,E1 -18782.494,E2 -18782.494} C_VEL
LIN {X 0,Y 260.855,Z 156.079,A -85,B 0,C 180,E1 -18783.206,E2 -18783.206} C_VEL
LIN {X 0,Y 259.272,Z 210.992,A -85,B 0,C 180,E1 -18784.727,E2 -18784.727} C_VEL
LIN {X 0,Y 258.361,Z 224.04,A -85,B 0,C 180,E1 -18785.384,E2 -18785.384} C_VEL
LIN {X 0,Y 257,Z 236.646,A -85,B 0,C 180,E1 -18786.318,E2 -18786.318} C_VEL
LIN {X 0,Y 255.405,Z 248.664,A -85,B 0,C 180,E1 -18787.554,E2 -18787.554} C_VEL
LIN {X 0,Y 253.671,Z 260.192,A -85,B 0,C 180,E1 -18789.102,E2 -18789.102} C_VEL
LIN {X 0,Y 252.098,Z 270.597,A -85,B 0,C 180,E1 -18790.879,E2 -18790.879} C_VEL
LIN {X 0,Y 250.347,Z 280.893,A -85,B 0,C 180,E1 -18793.107,E2 -18793.107} C_VEL
LIN {X 0,Y 249.158,Z 288.98,A -85,B 0,C 180,E1 -18795.294,E2 -18795.294} C_VEL
LIN {X 0,Y 248.034,Z 296.255,A -85,B 0,C 180,E1 -18797.73,E2 -18797.73} C_VEL
LIN {X 0,Y 247.431,Z 302.057,A -85,B 0,C 180,E1 -18800.187,E2 -18800.187} C_VEL
LIN {X 0,Y 247.093,Z 306.611,A -85,B 0,C 180,E1 -18802.646,E2 -18802.646} C_VEL
LIN {X 0,Y 247.06,Z 310.061,A -85,B 0,C 180,E1 -18805.104,E2 -18805.104} C_VEL
LIN {X 0,Y 247.138,Z 311.768,A -85,B 0,C 180,E1 -18806.739,E2 -18806.739} C_VEL
LIN {X 0,Y 247.166,Z 313.055,A -85,B 0,C 180,E1 -18808.37,E2 -18808.37} C_VEL
LIN {X 0,Y 247.223,Z 313.939,A -85,B 0,C 180,E1 -18810,E2 -18810} C_VEL
LIN {X 0,Y 247.109,Z 314.382,A -85,B 0,C 180,E1 -18811.63,E2 -18811.63} C_VEL
LIN {X 0,Y 247.052,Z 314.41,A -85,B 0,C 180,E1 -18813.261,E2 -18813.261} C_VEL
LIN {X 0,Y 246.991,Z 313.956,A -85,B 0,C 180,E1 -18815.182,E2 -18815.182} C_VEL
LIN {X 0,Y 247.172,Z 312.157,A -85,B 0,C 180,E1 -18818.173,E2 -18818.173} C_VEL
LIN {X 0,Y 247.518,Z 310.572,A -85,B 0,C 180,E1 -18819.809,E2 -18819.809} C_VEL
LIN {X 0,Y 248.25,Z 307.423,A -85,B 0,C 180,E1 -18822.259,E2 -18822.259} C_VEL
LIN {X 0,Y 249.554,Z 303.245,A -85,B 0,C 180,E1 -18824.682,E2 -18824.682} C_VEL
LIN {X 0,Y 251.633,Z 296.905,A -85,B 0,C 180,E1 -18827.472,E2 -18827.472} C_VEL
LIN {X 0,Y 253.76,Z 290.036,A -85,B 0,C 180,E1 -18829.832,E2 -18829.832} C_VEL
LIN {X 0,Y 256.413,Z 281.507,A -85,B 0,C 180,E1 -18832.14,E2 -18832.14} C_VEL
LIN {X 0,Y 259.087,Z 272.772,A -85,B 0,C 180,E1 -18834.01,E2 -18834.01} C_VEL
LIN {X 0,Y 262.034,Z 262.048,A -85,B 0,C 180,E1 -18835.839,E2 -18835.839} C_VEL
LIN {X 0,Y 264.653,Z 251.378,A -85,B 0,C 180,E1 -18837.264,E2 -18837.264} C_VEL
LIN {X 0,Y 267.099,Z 239.44,A -85,B 0,C 180,E1 -18838.484,E2 -18838.484} C_VEL
LIN {X 0,Y 269.159,Z 227.032,A -85,B 0,C 180,E1 -18839.42,E2 -18839.42} C_VEL
LIN {X 0,Y 270.63,Z 213.869,A -85,B 0,C 180,E1 -18840.12,E2 -18840.12} C_VEL
LIN {X 0,Y 271.588,Z 199.488,A -85,B 0,C 180,E1 -18840.557,E2 -18840.557} C_VEL
LIN {X 0,Y 273.071,Z 158.89,A -85,B 0,C 180,E1 -18841.624,E2 -18841.624} C_VEL
LIN {X 0,Y 269.685,Z 136.562,A -85,B 0,C 180,E1 -18842.861,E2 -18842.861} C_VEL
LIN {X 0,Y 267.911,Z 127.952,A -85,B 0,C 180,E1 -18843.428,E2 -18843.428} C_VEL
LIN {X 0,Y 260.908,Z 112.818,A -85,B 0,C 180,E1 -18845.127,E2 -18845.127} C_VEL
LIN {X 0,Y 255.794,Z 103.11,A -85,B 0,C 180,E1 -18846.408,E2 -18846.408} C_VEL
LIN {X 0,Y 253.976,Z 99.246,A -85,B 0,C 180,E1 -18846.923,E2 -18846.923} C_VEL
LIN {X 0,Y 251.954,Z 91.538,A -85,B 0,C 180,E1 -18850.3,E2 -18850.3} C_VEL
LIN {X 0,Y 249.671,Z 83.624,A -85,B 0,C 180,E1 -18854.07,E2 -18854.07} C_VEL
LIN {X 0,Y 249.03,Z 81.456,A -85,B 0,C 180,E1 -18855.268,E2 -18855.268} C_VEL
LIN {X 0,Y 249.009,Z 81.456,A -85,B 0,C 180,E1 -18859.645,E2 -18859.645} C_VEL
LIN {X 0,Y 249.032,Z 81.454,A -85,B 0,C 180,E1 -18863.655,E2 -18863.655} C_VEL
LIN {X 0,Y 249.04,Z 81.462,A -85,B 0,C 180,E1 -18867.845,E2 -18867.845} C_VEL
LIN {X 0,Y 249.1,Z 81.453,A -85,B 0,C 180,E1 -18871.338,E2 -18871.338} C_VEL
LIN {X 0,Y 249.154,Z 81.442,A -85,B 0,C 180,E1 -18874.969,E2 -18874.969} C_VEL
LIN {X 0,Y 249.114,Z 81.453,A -85,B 0,C 180,E1 -18880.212,E2 -18880.212} C_VEL
LIN {X 0,Y 249.245,Z 81.427,A -85,B 0,C 180,E1 -18883.622,E2 -18883.622} C_VEL
LIN {X 0,Y 249.248,Z 81.426,A -85,B 0,C 180,E1 -18888.616,E2 -18888.616} C_VEL
LIN {X 0,Y 249.458,Z 81.402,A -85,B 0,C 180,E1 -18891.902,E2 -18891.902} C_VEL
LIN {X 0,Y 249.296,Z 81.43,A -85,B 0,C 180,E1 -18895.148,E2 -18895.148} C_VEL
LIN {X 0,Y 249.677,Z 81.369,A -85,B 0,C 180,E1 -18898.387,E2 -18898.387} C_VEL
LIN {X 0,Y 249.678,Z 81.383,A -85,B 0,C 180,E1 -18901.613,E2 -18901.613} C_VEL
LIN {X 0,Y 249.437,Z 81.411,A -85,B 0,C 180,E1 -18906.69,E2 -18906.69} C_VEL
LIN {X 0,Y 249.345,Z 81.414,A -85,B 0,C 180,E1 -18909.736,E2 -18909.736} C_VEL
LIN {X 0,Y 249.185,Z 81.435,A -85,B 0,C 180,E1 -18914.704,E2 -18914.704} C_VEL
LIN {X 0,Y 249.123,Z 81.443,A -85,B 0,C 180,E1 -18918.078,E2 -18918.078} C_VEL
LIN {X 0,Y 249.086,Z 81.456,A -85,B 0,C 180,E1 -18921.518,E2 -18921.518} C_VEL
LIN {X 0,Y 249.108,Z 81.455,A -85,B 0,C 180,E1 -18925.47,E2 -18925.47} C_VEL
LIN {X 0,Y 249.043,Z 81.464,A -85,B 0,C 180,E1 -18928.976,E2 -18928.976} C_VEL
LIN {X 0,Y 249.028,Z 81.467,A -85,B 0,C 180,E1 -18932.426,E2 -18932.426} C_VEL
LIN {X 0,Y 249.028,Z 81.462,A -85,B 0,C 180,E1 -18936.346,E2 -18936.346} C_VEL
LIN {X 0,Y 249.006,Z 81.448,A -85,B 0,C 180,E1 -18940.478,E2 -18940.478} C_VEL
LIN {X 0,Y 249.032,Z 81.479,A -85,B 0,C 180,E1 -18942.223,E2 -18942.223} C_VEL
LIN {X 0,Y 249.934,Z 84.131,A -85,B 0,C 180,E1 -18942.512,E2 -18942.512} C_VEL
LIN {X 0,Y 252.063,Z 86.965,A -85,B 0,C 180,E1 -18943.054,E2 -18943.054} C_VEL
LIN {X 0,Y 260.407,Z 99.973,A -85,B 0,C 180,E1 -18945.12,E2 -18945.12} C_VEL
LIN {X 0,Y 267.302,Z 111.69,A -85,B 0,C 180,E1 -18946.716,E2 -18946.716} C_VEL
LIN {X 0,Y 274.397,Z 126.685,A -85,B 0,C 180,E1 -18948.337,E2 -18948.337} C_VEL
LIN {X 0,Y 271.894,Z 185.081,A -85,B 0,C 180,E1 -18949.865,E2 -18949.865} C_VEL
LIN {X 0,Y 270.786,Z 198.539,A -85,B 0,C 180,E1 -18950.515,E2 -18950.515} C_VEL
LIN {X 0,Y 269.409,Z 210.876,A -85,B 0,C 180,E1 -18951.418,E2 -18951.418} C_VEL
LIN {X 0,Y 267.552,Z 221.972,A -85,B 0,C 180,E1 -18952.484,E2 -18952.484} C_VEL
LIN {X 0,Y 265.259,Z 233.125,A -85,B 0,C 180,E1 -18953.877,E2 -18953.877} C_VEL
LIN {X 0,Y 262.709,Z 243.848,A -85,B 0,C 180,E1 -18955.588,E2 -18955.588} C_VEL
LIN {X 0,Y 260.275,Z 252.549,A -85,B 0,C 180,E1 -18957.313,E2 -18957.313} C_VEL
LIN {X 0,Y 257.82,Z 260.513,A -85,B 0,C 180,E1 -18959.262,E2 -18959.262} C_VEL
LIN {X 0,Y 255.63,Z 267.314,A -85,B 0,C 180,E1 -18961.331,E2 -18961.331} C_VEL
LIN {X 0,Y 253.426,Z 273.451,A -85,B 0,C 180,E1 -18963.659,E2 -18963.659} C_VEL
LIN {X 0,Y 251.559,Z 278.471,A -85,B 0,C 180,E1 -18966.103,E2 -18966.103} C_VEL
LIN {X 0,Y 250.075,Z 282.315,A -85,B 0,C 180,E1 -18968.571,E2 -18968.571} C_VEL
LIN {X 0,Y 249.233,Z 284.276,A -85,B 0,C 180,E1 -18970.222,E2 -18970.222} C_VEL
LIN {X 0,Y 248.558,Z 285.811,A -85,B 0,C 180,E1 -18971.879,E2 -18971.879} C_VEL
LIN {X 0,Y 247.782,Z 287.391,A -85,B 0,C 180,E1 -18974.658,E2 -18974.658} C_VEL
LIN {X 0,Y 247.354,Z 287.809,A -85,B 0,C 180,E1 -18976.862,E2 -18976.862} C_VEL
LIN {X 0,Y 247.104,Z 287.689,A -85,B 0,C 180,E1 -18978.516,E2 -18978.516} C_VEL
LIN {X 0,Y 247.054,Z 287.125,A -85,B 0,C 180,E1 -18980.173,E2 -18980.173} C_VEL
LIN {X 0,Y 247.344,Z 284.806,A -85,B 0,C 180,E1 -18983.474,E2 -18983.474} C_VEL
LIN {X 0,Y 247.589,Z 281.973,A -85,B 0,C 180,E1 -18985.931,E2 -18985.931} C_VEL
LIN {X 0,Y 248.094,Z 278.122,A -85,B 0,C 180,E1 -18988.377,E2 -18988.377} C_VEL
LIN {X 0,Y 248.704,Z 273.165,A -85,B 0,C 180,E1 -18990.81,E2 -18990.81} C_VEL
LIN {X 0,Y 249.748,Z 266.927,A -85,B 0,C 180,E1 -18993.227,E2 -18993.227} C_VEL
LIN {X 0,Y 251.077,Z 259.124,A -85,B 0,C 180,E1 -18995.622,E2 -18995.622} C_VEL
LIN {X 0,Y 252.68,Z 249.405,A -85,B 0,C 180,E1 -18997.994,E2 -18997.994} C_VEL
LIN {X 0,Y 254.254,Z 240.395,A -85,B 0,C 180,E1 -18999.748,E2 -18999.748} C_VEL
LIN {X 0,Y 256.008,Z 229.223,A -85,B 0,C 180,E1 -19001.48,E2 -19001.48} C_VEL
LIN {X 0,Y 257.392,Z 218.313,A -85,B 0,C 180,E1 -19002.818,E2 -19002.818} C_VEL
LIN {X 0,Y 258.524,Z 206.29,A -85,B 0,C 180,E1 -19003.962,E2 -19003.962} C_VEL
LIN {X 0,Y 259.42,Z 193.818,A -85,B 0,C 180,E1 -19004.814,E2 -19004.814} C_VEL
LIN {X 0,Y 260.02,Z 180.818,A -85,B 0,C 180,E1 -19005.38,E2 -19005.38} C_VEL
LIN {X 0,Y 261.978,Z 113.197,A -85,B 0,C 180,E1 -19007.202,E2 -19007.202} C_VEL
LIN {X 0,Y 260.973,Z 109.328,A -85,B 0,C 180,E1 -19007.413,E2 -19007.413} C_VEL
LIN {X 0,Y 256.981,Z 98.869,A -85,B 0,C 180,E1 -19008.121,E2 -19008.121} C_VEL
LIN {X 0,Y 249.245,Z 82.036,A -85,B 0,C 180,E1 -19009.461,E2 -19009.461} C_VEL
LIN {X 0,Y 249.128,Z 81.452,A -85,B 0,C 180,E1 -19009.586,E2 -19009.586} C_VEL
LIN {X 0,Y 249.063,Z 81.458,A -85,B 0,C 180,E1 -19013.269,E2 -19013.269} C_VEL
LIN {X 0,Y 249.07,Z 81.459,A -85,B 0,C 180,E1 -19016.839,E2 -19016.839} C_VEL
LIN {X 0,Y 249.049,Z 81.46,A -85,B 0,C 180,E1 -19020.528,E2 -19020.528} C_VEL
LIN {X 0,Y 249.076,Z 81.457,A -85,B 0,C 180,E1 -19025.088,E2 -19025.088} C_VEL
LIN {X 0,Y 249.041,Z 81.462,A -85,B 0,C 180,E1 -19028.378,E2 -19028.378} C_VEL
LIN {X 0,Y 249.014,Z 81.464,A -85,B 0,C 180,E1 -19032.794,E2 -19032.794} C_VEL
LIN {X 0,Y 249.011,Z 81.468,A -85,B 0,C 180,E1 -19037.362,E2 -19037.362} C_VEL
LIN {X 0,Y 249.028,Z 81.464,A -85,B 0,C 180,E1 -19041.62,E2 -19041.62} C_VEL
LIN {X 0,Y 249.046,Z 81.461,A -85,B 0,C 180,E1 -19045.64,E2 -19045.64} C_VEL
LIN {X 0,Y 249.054,Z 81.457,A -85,B 0,C 180,E1 -19049.474,E2 -19049.474} C_VEL
LIN {X 0,Y 249.076,Z 81.458,A -85,B 0,C 180,E1 -19053.163,E2 -19053.163} C_VEL
